LIN {X 0,Y 500.649,Z 462.149,A -85,B 0,C 180,E1 12941.575,E2 12941.575} C_VEL
LIN {X 0,Y 506.783,Z 470.16,A -85,B 0,C 180,E1 12939.56,E2 12939.56} C_VEL
LIN {X 0,Y 513.337,Z 479.72,A -85,B 0,C 180,E1 12937.586,E2 12937.586} C_VEL
LIN {X 0,Y 523.821,Z 496.267,A -85,B 0,C 180,E1 12934.746,E2 12934.746} C_VEL
LIN {X 0,Y 529.057,Z 505.232,A -85,B 0,C 180,E1 12933.44,E2 12933.44} C_VEL
LIN {X 0,Y 516.289,Z 720.849,A -85,B 0,C 180,E1 12930.101,E2 12930.101} C_VEL
LIN {X 0,Y 510.116,Z 825.661,A -85,B 0,C 180,E1 12928.464,E2 12928.464} C_VEL
LIN {X 0,Y 507.28,Z 853.259,A -85,B 0,C 180,E1 12927.934,E2 12927.934} C_VEL
LIN {X 0,Y 503.396,Z 879.439,A -85,B 0,C 180,E1 12927.252,E2 12927.252} C_VEL
LIN {X 0,Y 499.633,Z 900.65,A -85,B 0,C 180,E1 12926.565,E2 12926.565} C_VEL
LIN {X 0,Y 495.492,Z 920.963,A -85,B 0,C 180,E1 12925.777,E2 12925.777} C_VEL
LIN {X 0,Y 490.621,Z 942.152,A -85,B 0,C 180,E1 12924.809,E2 12924.809} C_VEL
LIN {X 0,Y 484.197,Z 967.245,A -85,B 0,C 180,E1 12923.446,E2 12923.446} C_VEL
LIN {X 0,Y 477.712,Z 989.541,A -85,B 0,C 180,E1 12922.003,E2 12922.003} C_VEL
LIN {X 0,Y 471.761,Z 1008.579,A -85,B 0,C 180,E1 12920.583,E2 12920.583} C_VEL
LIN {X 0,Y 465.626,Z 1027.087,A -85,B 0,C 180,E1 12919.009,E2 12919.009} C_VEL
LIN {X 0,Y 458.527,Z 1047.528,A -85,B 0,C 180,E1 12917.018,E2 12917.018} C_VEL
LIN {X 0,Y 450.725,Z 1068.736,A -85,B 0,C 180,E1 12914.593,E2 12914.593} C_VEL
LIN {X 0,Y 444.621,Z 1084.894,A -85,B 0,C 180,E1 12912.47,E2 12912.47} C_VEL
LIN {X 0,Y 438.714,Z 1100.381,A -85,B 0,C 180,E1 12910.165,E2 12910.165} C_VEL
LIN {X 0,Y 432.278,Z 1117.401,A -85,B 0,C 180,E1 12907.279,E2 12907.279} C_VEL
LIN {X 0,Y 426.222,Z 1133.289,A -85,B 0,C 180,E1 12904.103,E2 12904.103} C_VEL
LIN {X 0,Y 422.001,Z 1145.022,A -85,B 0,C 180,E1 12901.417,E2 12901.417} C_VEL
LIN {X 0,Y 418.256,Z 1156.002,A -85,B 0,C 180,E1 12898.563,E2 12898.563} C_VEL
LIN {X 0,Y 414.556,Z 1167.99,A -85,B 0,C 180,E1 12894.967,E2 12894.967} C_VEL
LIN {X 0,Y 411.822,Z 1177.9,A -85,B 0,C 180,E1 12891.358,E2 12891.358} C_VEL
LIN {X 0,Y 410.259,Z 1184.648,A -85,B 0,C 180,E1 12888.472,E2 12888.472} C_VEL
LIN {X 0,Y 409.201,Z 1190.344,A -85,B 0,C 180,E1 12885.592,E2 12885.592} C_VEL
LIN {X 0,Y 408.507,Z 1195.031,A -85,B 0,C 180,E1 12882.726,E2 12882.726} C_VEL
LIN {X 0,Y 408.142,Z 1198.741,A -85,B 0,C 180,E1 12879.875,E2 12879.875} C_VEL
LIN {X 0,Y 407.972,Z 1201.501,A -85,B 0,C 180,E1 12877.039,E2 12877.039} C_VEL
LIN {X 0,Y 407.917,Z 1203.331,A -85,B 0,C 180,E1 12874.218,E2 12874.218} C_VEL
LIN {X 0,Y 407.911,Z 1204.221,A -85,B 0,C 180,E1 12871.546,E2 12871.546} C_VEL
LIN {X 0,Y 407.912,Z 1204.288,A -85,B 0,C 180,E1 12868.877,E2 12868.877} C_VEL
LIN {X 0,Y 407.916,Z 1203.463,A -85,B 0,C 180,E1 12866.065,E2 12866.065} C_VEL
LIN {X 0,Y 407.964,Z 1201.721,A -85,B 0,C 180,E1 12863.244,E2 12863.244} C_VEL
LIN {X 0,Y 408.116,Z 1199.054,A -85,B 0,C 180,E1 12860.41,E2 12860.41} C_VEL
LIN {X 0,Y 408.484,Z 1195.239,A -85,B 0,C 180,E1 12857.418,E2 12857.418} C_VEL
LIN {X 0,Y 409.157,Z 1190.625,A -85,B 0,C 180,E1 12854.552,E2 12854.552} C_VEL
LIN {X 0,Y 410.263,Z 1184.721,A -85,B 0,C 180,E1 12851.529,E2 12851.529} C_VEL
LIN {X 0,Y 412.02,Z 1177.346,A -85,B 0,C 180,E1 12848.355,E2 12848.355} C_VEL
LIN {X 0,Y 415.114,Z 1166.541,A -85,B 0,C 180,E1 12844.46,E2 12844.46} C_VEL
LIN {X 0,Y 418.676,Z 1155.593,A -85,B 0,C 180,E1 12841.158,E2 12841.158} C_VEL
LIN {X 0,Y 422.528,Z 1144.786,A -85,B 0,C 180,E1 12838.309,E2 12838.309} C_VEL
LIN {X 0,Y 427.171,Z 1132.591,A -85,B 0,C 180,E1 12835.481,E2 12835.481} C_VEL
LIN {X 0,Y 433.755,Z 1116.189,A -85,B 0,C 180,E1 12832.182,E2 12832.182} C_VEL
LIN {X 0,Y 440.101,Z 1100.481,A -85,B 0,C 180,E1 12829.477,E2 12829.477} C_VEL
LIN {X 0,Y 446.32,Z 1085.225,A -85,B 0,C 180,E1 12827.163,E2 12827.163} C_VEL
LIN {X 0,Y 452.763,Z 1069.315,A -85,B 0,C 180,E1 12825.035,E2 12825.035} C_VEL
LIN {X 0,Y 460.874,Z 1048.953,A -85,B 0,C 180,E1 12822.654,E2 12822.654} C_VEL
LIN {X 0,Y 468.875,Z 1027.549,A -85,B 0,C 180,E1 12820.538,E2 12820.538} C_VEL
LIN {X 0,Y 475.563,Z 1008.838,A -85,B 0,C 180,E1 12818.93,E2 12818.93} C_VEL
LIN {X 0,Y 482.02,Z 989.698,A -85,B 0,C 180,E1 12817.493,E2 12817.493} C_VEL
LIN {X 0,Y 489.336,Z 966.442,A -85,B 0,C 180,E1 12815.987,E2 12815.987} C_VEL
LIN {X 0,Y 496.05,Z 942.158,A -85,B 0,C 180,E1 12814.676,E2 12814.676} C_VEL
LIN {X 0,Y 501.27,Z 921.153,A -85,B 0,C 180,E1 12813.719,E2 12813.719} C_VEL
LIN {X 0,Y 505.768,Z 900.797,A -85,B 0,C 180,E1 12812.934,E2 12812.934} C_VEL
LIN {X 0,Y 509.793,Z 879.827,A -85,B 0,C 180,E1 12812.258,E2 12812.258} C_VEL
LIN {X 0,Y 513.643,Z 855.953,A -85,B 0,C 180,E1 12811.636,E2 12811.636} C_VEL
LIN {X 0,Y 517.066,Z 826.781,A -85,B 0,C 180,E1 12811.063,E2 12811.063} C_VEL
LIN {X 0,Y 521.805,Z 756.676,A -85,B 0,C 180,E1 12809.953,E2 12809.953} C_VEL
LIN {X 0,Y 536.543,Z 536.341,A -85,B 0,C 180,E1 12806.519,E2 12806.519} C_VEL
LIN {X 0,Y 538.44,Z 508.698,A -85,B 0,C 180,E1 12806.082,E2 12806.082} C_VEL
LIN {X 0,Y 531.522,Z 497.374,A -85,B 0,C 180,E1 12803.91,E2 12803.91} C_VEL
LIN {X 0,Y 523.953,Z 485.597,A -85,B 0,C 180,E1 12801.201,E2 12801.201} C_VEL
LIN {X 0,Y 519.684,Z 479.746,A -85,B 0,C 180,E1 12799.481,E2 12799.481} C_VEL
LIN {X 0,Y 516.251,Z 475.069,A -85,B 0,C 180,E1 12797.936,E2 12797.936} C_VEL
LIN {X 0,Y 512.607,Z 470.139,A -85,B 0,C 180,E1 12796.08,E2 12796.08} C_VEL
LIN {X 0,Y 508.761,Z 464.995,A -85,B 0,C 180,E1 12793.757,E2 12793.757} C_VEL
LIN {X 0,Y 505.748,Z 461.392,A -85,B 0,C 180,E1 12791.518,E2 12791.518} C_VEL
LIN {X 0,Y 504.696,Z 459.401,A -85,B 0,C 180,E1 12790.502,E2 12790.502} C_VEL
LIN {X 0,Y 501.449,Z 455.939,A -85,B 0,C 180,E1 12786.181,E2 12786.181} C_VEL
LIN {X 0,Y 500.926,Z 453.438,A -85,B 0,C 180,E1 12783.319,E2 12783.319} C_VEL
LIN {X 0,Y 500.952,Z 453.714,A -85,B 0,C 180,E1 12781.945,E2 12781.945} C_VEL
LIN {X 0,Y 503.821,Z 458.829,A -85,B 0,C 180,E1 12776.131,E2 12776.131} C_VEL
LIN {X 0,Y 504.993,Z 459.862,A -85,B 0,C 180,E1 12775.002,E2 12775.002} C_VEL
LIN {X 0,Y 507.681,Z 463.98,A -85,B 0,C 180,E1 12772.759,E2 12772.759} C_VEL
LIN {X 0,Y 509.358,Z 465.743,A -85,B 0,C 180,E1 12771.647,E2 12771.647} C_VEL
LIN {X 0,Y 512.705,Z 470.216,A -85,B 0,C 180,E1 12769.664,E2 12769.664} C_VEL
LIN {X 0,Y 517.641,Z 476.786,A -85,B 0,C 180,E1 12767.222,E2 12767.222} C_VEL
LIN {X 0,Y 522.414,Z 483.411,A -85,B 0,C 180,E1 12765.196,E2 12765.196} C_VEL
LIN {X 0,Y 527.766,Z 490.712,A -85,B 0,C 180,E1 12763.206,E2 12763.206} C_VEL
LIN {X 0,Y 535.807,Z 502.584,A -85,B 0,C 180,E1 12760.571,E2 12760.571} C_VEL
LIN {X 0,Y 538.454,Z 506.775,A -85,B 0,C 180,E1 12759.773,E2 12759.773} C_VEL
LIN {X 0,Y 524.368,Z 714.828,A -85,B 0,C 180,E1 12756.529,E2 12756.529} C_VEL
LIN {X 0,Y 517.356,Z 819.989,A -85,B 0,C 180,E1 12754.874,E2 12754.874} C_VEL
LIN {X 0,Y 514.276,Z 847.618,A -85,B 0,C 180,E1 12754.34,E2 12754.34} C_VEL
LIN {X 0,Y 510.217,Z 873.27,A -85,B 0,C 180,E1 12753.669,E2 12753.669} C_VEL
LIN {X 0,Y 506.139,Z 894.675,A -85,B 0,C 180,E1 12752.975,E2 12752.975} C_VEL
LIN {X 0,Y 501.675,Z 915.064,A -85,B 0,C 180,E1 12752.18,E2 12752.18} C_VEL
LIN {X 0,Y 496.561,Z 935.717,A -85,B 0,C 180,E1 12751.232,E2 12751.232} C_VEL
LIN {X 0,Y 489.92,Z 959.881,A -85,B 0,C 180,E1 12749.92,E2 12749.92} C_VEL
LIN {X 0,Y 482.807,Z 982.517,A -85,B 0,C 180,E1 12748.451,E2 12748.451} C_VEL
LIN {X 0,Y 476.282,Z 1001.817,A -85,B 0,C 180,E1 12747,E2 12747} C_VEL
LIN {X 0,Y 469.809,Z 1019.855,A -85,B 0,C 180,E1 12745.449,E2 12745.449} C_VEL
LIN {X 0,Y 462.48,Z 1039.301,A -85,B 0,C 180,E1 12743.538,E2 12743.538} C_VEL
LIN {X 0,Y 453.885,Z 1060.944,A -85,B 0,C 180,E1 12741.043,E2 12741.043} C_VEL
LIN {X 0,Y 447.252,Z 1077.112,A -85,B 0,C 180,E1 12738.884,E2 12738.884} C_VEL
LIN {X 0,Y 441.031,Z 1092.119,A -85,B 0,C 180,E1 12736.61,E2 12736.61} C_VEL
LIN {X 0,Y 434.761,Z 1107.334,A -85,B 0,C 180,E1 12733.99,E2 12733.99} C_VEL
LIN {X 0,Y 427.725,Z 1124.554,A -85,B 0,C 180,E1 12730.531,E2 12730.531} C_VEL
LIN {X 0,Y 423.052,Z 1136.488,A -85,B 0,C 180,E1 12727.744,E2 12727.744} C_VEL
LIN {X 0,Y 419.137,Z 1147.1,A -85,B 0,C 180,E1 12724.926,E2 12724.926} C_VEL
LIN {X 0,Y 415.741,Z 1157.091,A -85,B 0,C 180,E1 12721.897,E2 12721.897} C_VEL
LIN {X 0,Y 412.5,Z 1167.903,A -85,B 0,C 180,E1 12718.05,E2 12718.05} C_VEL
LIN {X 0,Y 410.47,Z 1175.834,A -85,B 0,C 180,E1 12714.616,E2 12714.616} C_VEL
LIN {X 0,Y 409.314,Z 1181.594,A -85,B 0,C 180,E1 12711.645,E2 12711.645} C_VEL
LIN {X 0,Y 408.567,Z 1186.304,A -85,B 0,C 180,E1 12708.698,E2 12708.698} C_VEL
LIN {X 0,Y 408.177,Z 1190.004,A -85,B 0,C 180,E1 12705.777,E2 12705.777} C_VEL
LIN {X 0,Y 407.984,Z 1192.727,A -85,B 0,C 180,E1 12702.886,E2 12702.886} C_VEL
LIN {X 0,Y 407.921,Z 1194.501,A -85,B 0,C 180,E1 12700.022,E2 12700.022} C_VEL
LIN {X 0,Y 407.919,Z 1195.326,A -85,B 0,C 180,E1 12697.322,E2 12697.322} C_VEL
LIN {X 0,Y 407.905,Z 1195.359,A -85,B 0,C 180,E1 12694.803,E2 12694.803} C_VEL
LIN {X 0,Y 406.92,Z 1195.204,A -85,B 0,C 180,E1 12693.721,E2 12693.721} C_VEL
LIN {X 0,Y 401.978,Z 1194.558,A -85,B 0,C 180,E1 12691.527,E2 12691.527} C_VEL
LIN {X 0,Y 400.057,Z 1193.818,A -85,B 0,C 180,E1 12690.199,E2 12690.199} C_VEL
LIN {X 0,Y 399.972,Z 1193.575,A -85,B 0,C 180,E1 12689.88,E2 12689.88} C_VEL
LIN {X 0,Y 400.145,Z 1190.587,A -85,B 0,C 180,E1 12686.418,E2 12686.418} C_VEL
LIN {X 0,Y 400.568,Z 1186.761,A -85,B 0,C 180,E1 12683.262,E2 12683.262} C_VEL
LIN {X 0,Y 401.314,Z 1182.083,A -85,B 0,C 180,E1 12680.245,E2 12680.245} C_VEL
LIN {X 0,Y 402.511,Z 1176.366,A -85,B 0,C 180,E1 12677.227,E2 12677.227} C_VEL
LIN {X 0,Y 404.331,Z 1169.229,A -85,B 0,C 180,E1 12674.068,E2 12674.068} C_VEL
LIN {X 0,Y 407.469,Z 1158.801,A -85,B 0,C 180,E1 12670.206,E2 12670.206} C_VEL
LIN {X 0,Y 411.238,Z 1147.66,A -85,B 0,C 180,E1 12666.792,E2 12666.792} C_VEL
LIN {X 0,Y 415.137,Z 1136.992,A -85,B 0,C 180,E1 12663.949,E2 12663.949} C_VEL
LIN {X 0,Y 419.622,Z 1125.365,A -85,B 0,C 180,E1 12661.227,E2 12661.227} C_VEL
LIN {X 0,Y 425.801,Z 1110.09,A -85,B 0,C 180,E1 12658.105,E2 12658.105} C_VEL
LIN {X 0,Y 432.54,Z 1093.213,A -85,B 0,C 180,E1 12655.181,E2 12655.181} C_VEL
LIN {X 0,Y 438.402,Z 1078.627,A -85,B 0,C 180,E1 12652.965,E2 12652.965} C_VEL
LIN {X 0,Y 444.443,Z 1063.364,A -85,B 0,C 180,E1 12650.911,E2 12650.911} C_VEL
LIN {X 0,Y 450.831,Z 1046.832,A -85,B 0,C 180,E1 12648.946,E2 12648.946} C_VEL
LIN {X 0,Y 458.984,Z 1024.761,A -85,B 0,C 180,E1 12646.668,E2 12646.668} C_VEL
LIN {X 0,Y 465.894,Z 1004.728,A -85,B 0,C 180,E1 12644.909,E2 12644.909} C_VEL
LIN {X 0,Y 471.704,Z 986.875,A -85,B 0,C 180,E1 12643.536,E2 12643.536} C_VEL
LIN {X 0,Y 477.203,Z 968.666,A -85,B 0,C 180,E1 12642.299,E2 12642.299} C_VEL
LIN {X 0,Y 482.904,Z 948.204,A -85,B 0,C 180,E1 12641.089,E2 12641.089} C_VEL
LIN {X 0,Y 489.102,Z 923.711,A -85,B 0,C 180,E1 12639.857,E2 12639.857} C_VEL
LIN {X 0,Y 494.568,Z 898.087,A -85,B 0,C 180,E1 12638.81,E2 12638.81} C_VEL
LIN {X 0,Y 498.547,Z 876.437,A -85,B 0,C 180,E1 12638.082,E2 12638.082} C_VEL
LIN {X 0,Y 501.804,Z 855.388,A -85,B 0,C 180,E1 12637.5,E2 12637.5} C_VEL
LIN {X 0,Y 504.663,Z 832.536,A -85,B 0,C 180,E1 12636.999,E2 12636.999} C_VEL
LIN {X 0,Y 507.414,Z 797.216,A -85,B 0,C 180,E1 12636.402,E2 12636.402} C_VEL
LIN {X 0,Y 520.73,Z 575.134,A -85,B 0,C 180,E1 12632.96,E2 12632.96} C_VEL
LIN {X 0,Y 524.893,Z 506.946,A -85,B 0,C 180,E1 12631.884,E2 12631.884} C_VEL
LIN {X 0,Y 515.61,Z 493.078,A -85,B 0,C 180,E1 12629.475,E2 12629.475} C_VEL
LIN {X 0,Y 507.533,Z 481.415,A -85,B 0,C 180,E1 12627.134,E2 12627.134} C_VEL
LIN {X 0,Y 499.579,Z 470.522,A -85,B 0,C 180,E1 12624.539,E2 12624.539} C_VEL
LIN {X 0,Y 495.044,Z 464.466,A -85,B 0,C 180,E1 12622.881,E2 12622.881} C_VEL
LIN {X 0,Y 492.214,Z 460.736,A -85,B 0,C 180,E1 12621.761,E2 12621.761} C_VEL
LIN {X 0,Y 488.391,Z 455.782,A -85,B 0,C 180,E1 12620.118,E2 12620.118} C_VEL
LIN {X 0,Y 484.466,Z 450.681,A -85,B 0,C 180,E1 12618.221,E2 12618.221} C_VEL
LIN {X 0,Y 481.081,Z 446.451,A -85,B 0,C 180,E1 12616.357,E2 12616.357} C_VEL
LIN {X 0,Y 480.021,Z 445.116,A -85,B 0,C 180,E1 12615.711,E2 12615.711} C_VEL
LIN {X 0,Y 476.73,Z 441.248,A -85,B 0,C 180,E1 12613.463,E2 12613.463} C_VEL
LIN {X 0,Y 475.75,Z 439.436,A -85,B 0,C 180,E1 12612.626,E2 12612.626} C_VEL
LIN {X 0,Y 472.527,Z 436.477,A -85,B 0,C 180,E1 12609.5,E2 12609.5} C_VEL
LIN {X 0,Y 471.237,Z 433.403,A -85,B 0,C 180,E1 12607.314,E2 12607.314} C_VEL
LIN {X 0,Y 470.236,Z 433.066,A -85,B 0,C 180,E1 12601.218,E2 12601.218} C_VEL
LIN {X 0,Y 471.366,Z 433.605,A -85,B 0,C 180,E1 12598.541,E2 12598.541} C_VEL
LIN {X 0,Y 473.121,Z 437.382,A -85,B 0,C 180,E1 12595.879,E2 12595.879} C_VEL
LIN {X 0,Y 476.09,Z 439.999,A -85,B 0,C 180,E1 12593.185,E2 12593.185} C_VEL
LIN {X 0,Y 479.035,Z 444.326,A -85,B 0,C 180,E1 12590.993,E2 12590.993} C_VEL
LIN {X 0,Y 480.77,Z 445.966,A -85,B 0,C 180,E1 12589.939,E2 12589.939} C_VEL
LIN {X 0,Y 484.188,Z 450.411,A -85,B 0,C 180,E1 12588.022,E2 12588.022} C_VEL
LIN {X 0,Y 485.549,Z 452.146,A -85,B 0,C 180,E1 12587.331,E2 12587.331} C_VEL
LIN {X 0,Y 490.234,Z 458.25,A -85,B 0,C 180,E1 12585.169,E2 12585.169} C_VEL
LIN {X 0,Y 494.275,Z 463.516,A -85,B 0,C 180,E1 12583.518,E2 12583.518} C_VEL
LIN {X 0,Y 499.024,Z 469.912,A -85,B 0,C 180,E1 12581.755,E2 12581.755} C_VEL
LIN {X 0,Y 504.843,Z 477.66,A -85,B 0,C 180,E1 12579.811,E2 12579.811} C_VEL
LIN {X 0,Y 511.142,Z 486.977,A -85,B 0,C 180,E1 12577.879,E2 12577.879} C_VEL
LIN {X 0,Y 521.2,Z 503.153,A -85,B 0,C 180,E1 12575.096,E2 12575.096} C_VEL
LIN {X 0,Y 524.916,Z 509.779,A -85,B 0,C 180,E1 12574.136,E2 12574.136} C_VEL
LIN {X 0,Y 511.66,Z 727.256,A -85,B 0,C 180,E1 12570.761,E2 12570.761} C_VEL
LIN {X 0,Y 505.683,Z 825.643,A -85,B 0,C 180,E1 12569.219,E2 12569.219} C_VEL
LIN {X 0,Y 502.773,Z 853.268,A -85,B 0,C 180,E1 12568.688,E2 12568.688} C_VEL
LIN {X 0,Y 498.795,Z 879.444,A -85,B 0,C 180,E1 12568.008,E2 12568.008} C_VEL
LIN {X 0,Y 495.004,Z 900.352,A -85,B 0,C 180,E1 12567.332,E2 12567.332} C_VEL
LIN {X 0,Y 490.612,Z 921.356,A -85,B 0,C 180,E1 12566.519,E2 12566.519} C_VEL
LIN {X 0,Y 485.516,Z 942.93,A -85,B 0,C 180,E1 12565.529,E2 12565.529} C_VEL
LIN {X 0,Y 478.478,Z 969.334,A -85,B 0,C 180,E1 12564.073,E2 12564.073} C_VEL
LIN {X 0,Y 472.363,Z 989.767,A -85,B 0,C 180,E1 12562.741,E2 12562.741} C_VEL
LIN {X 0,Y 466.248,Z 1008.785,A -85,B 0,C 180,E1 12561.316,E2 12561.316} C_VEL
LIN {X 0,Y 459.936,Z 1027.265,A -85,B 0,C 180,E1 12559.735,E2 12559.735} C_VEL
LIN {X 0,Y 452.09,Z 1049.172,A -85,B 0,C 180,E1 12557.579,E2 12557.579} C_VEL
LIN {X 0,Y 444.34,Z 1069.399,A -85,B 0,C 180,E1 12555.224,E2 12555.224} C_VEL
LIN {X 0,Y 438.024,Z 1085.545,A -85,B 0,C 180,E1 12553.074,E2 12553.074} C_VEL
LIN {X 0,Y 431.946,Z 1100.916,A -85,B 0,C 180,E1 12550.752,E2 12550.752} C_VEL
LIN {X 0,Y 425.025,Z 1118.465,A -85,B 0,C 180,E1 12547.71,E2 12547.71} C_VEL
LIN {X 0,Y 419.256,Z 1133.037,A -85,B 0,C 180,E1 12544.75,E2 12544.75} C_VEL
LIN {X 0,Y 414.815,Z 1144.793,A -85,B 0,C 180,E1 12542.026,E2 12542.026} C_VEL
LIN {X 0,Y 411.076,Z 1155.274,A -85,B 0,C 180,E1 12539.269,E2 12539.269} C_VEL
LIN {X 0,Y 407.531,Z 1165.97,A -85,B 0,C 180,E1 12536.052,E2 12536.052} C_VEL
LIN {X 0,Y 404.29,Z 1177.031,A -85,B 0,C 180,E1 12532.082,E2 12532.082} C_VEL
LIN {X 0,Y 402.43,Z 1184.512,A -85,B 0,C 180,E1 12528.845,E2 12528.845} C_VEL
LIN {X 0,Y 401.292,Z 1190.255,A -85,B 0,C 180,E1 12525.889,E2 12525.889} C_VEL
LIN {X 0,Y 400.553,Z 1194.921,A -85,B 0,C 180,E1 12522.983,E2 12522.983} C_VEL
LIN {X 0,Y 400.16,Z 1198.641,A -85,B 0,C 180,E1 12520.074,E2 12520.074} C_VEL
LIN {X 0,Y 399.98,Z 1201.407,A -85,B 0,C 180,E1 12517.181,E2 12517.181} C_VEL
LIN {X 0,Y 399.919,Z 1203.172,A -85,B 0,C 180,E1 12514.446,E2 12514.446} C_VEL
LIN {X 0,Y 399.91,Z 1204.11,A -85,B 0,C 180,E1 12511.72,E2 12511.72} C_VEL
LIN {X 0,Y 399.913,Z 1204.201,A -85,B 0,C 180,E1 12508.854,E2 12508.854} C_VEL
LIN {X 0,Y 399.916,Z 1203.378,A -85,B 0,C 180,E1 12505.986,E2 12505.986} C_VEL
LIN {X 0,Y 399.967,Z 1201.639,A -85,B 0,C 180,E1 12503.109,E2 12503.109} C_VEL
LIN {X 0,Y 400.134,Z 1198.977,A -85,B 0,C 180,E1 12500.217,E2 12500.217} C_VEL
LIN {X 0,Y 400.529,Z 1195.171,A -85,B 0,C 180,E1 12497.164,E2 12497.164} C_VEL
LIN {X 0,Y 401.256,Z 1190.568,A -85,B 0,C 180,E1 12494.24,E2 12494.24} C_VEL
LIN {X 0,Y 402.439,Z 1184.677,A -85,B 0,C 180,E1 12491.157,E2 12491.157} C_VEL
LIN {X 0,Y 404.211,Z 1177.673,A -85,B 0,C 180,E1 12488.068,E2 12488.068} C_VEL
LIN {X 0,Y 407.315,Z 1167.462,A -85,B 0,C 180,E1 12484.247,E2 12484.247} C_VEL
LIN {X 0,Y 411.36,Z 1155.619,A -85,B 0,C 180,E1 12480.595,E2 12480.595} C_VEL
LIN {X 0,Y 415.404,Z 1144.835,A -85,B 0,C 180,E1 12477.701,E2 12477.701} C_VEL
LIN {X 0,Y 420.266,Z 1132.729,A -85,B 0,C 180,E1 12474.848,E2 12474.848} C_VEL
LIN {X 0,Y 426.858,Z 1117.069,A -85,B 0,C 180,E1 12471.631,E2 12471.631} C_VEL
LIN {X 0,Y 434.127,Z 1099.793,A -85,B 0,C 180,E1 12468.624,E2 12468.624} C_VEL
LIN {X 0,Y 440.595,Z 1084.568,A -85,B 0,C 180,E1 12466.306,E2 12466.306} C_VEL
LIN {X 0,Y 447.564,Z 1068.023,A -85,B 0,C 180,E1 12464.091,E2 12464.091} C_VEL
LIN {X 0,Y 456.708,Z 1045.635,A -85,B 0,C 180,E1 12461.519,E2 12461.519} C_VEL
LIN {X 0,Y 463.896,Z 1027.059,A -85,B 0,C 180,E1 12459.694,E2 12459.694} C_VEL
LIN {X 0,Y 470.739,Z 1008.48,A -85,B 0,C 180,E1 12458.098,E2 12458.098} C_VEL
LIN {X 0,Y 477.478,Z 989.056,A -85,B 0,C 180,E1 12456.643,E2 12456.643} C_VEL
LIN {X 0,Y 485.246,Z 964.909,A -85,B 0,C 180,E1 12455.093,E2 12455.093} C_VEL
LIN {X 0,Y 491.829,Z 941.655,A -85,B 0,C 180,E1 12453.852,E2 12453.852} C_VEL
LIN {X 0,Y 497.181,Z 920.632,A -85,B 0,C 180,E1 12452.9,E2 12452.9} C_VEL
LIN {X 0,Y 501.767,Z 900.354,A -85,B 0,C 180,E1 12452.125,E2 12452.125} C_VEL
LIN {X 0,Y 505.982,Z 878.799,A -85,B 0,C 180,E1 12451.436,E2 12451.436} C_VEL
LIN {X 0,Y 510.346,Z 852.054,A -85,B 0,C 180,E1 12450.759,E2 12450.759} C_VEL
LIN {X 0,Y 513.404,Z 824.903,A -85,B 0,C 180,E1 12450.245,E2 12450.245} C_VEL
LIN {X 0,Y 523.571,Z 675.798,A -85,B 0,C 180,E1 12447.904,E2 12447.904} C_VEL
LIN {X 0,Y 534.88,Z 513.617,A -85,B 0,C 180,E1 12445.363,E2 12445.363} C_VEL
LIN {X 0,Y 529.15,Z 504.104,A -85,B 0,C 180,E1 12443.498,E2 12443.498} C_VEL
LIN {X 0,Y 522.018,Z 492.763,A -85,B 0,C 180,E1 12440.871,E2 12440.871} C_VEL
LIN {X 0,Y 518.002,Z 487.199,A -85,B 0,C 180,E1 12439.215,E2 12439.215} C_VEL
LIN {X 0,Y 514.708,Z 482.637,A -85,B 0,C 180,E1 12437.699,E2 12437.699} C_VEL
LIN {X 0,Y 511.234,Z 477.845,A -85,B 0,C 180,E1 12435.892,E2 12435.892} C_VEL
LIN {X 0,Y 507.454,Z 472.745,A -85,B 0,C 180,E1 12433.561,E2 12433.561} C_VEL
LIN {X 0,Y 504.457,Z 468.974,A -85,B 0,C 180,E1 12431.259,E2 12431.259} C_VEL
LIN {X 0,Y 503.607,Z 467.296,A -85,B 0,C 180,E1 12430.409,E2 12430.409} C_VEL
LIN {X 0,Y 500.383,Z 463.724,A -85,B 0,C 180,E1 12425.964,E2 12425.964} C_VEL
LIN {X 0,Y 499.95,Z 461.378,A -85,B 0,C 180,E1 12423.325,E2 12423.325} C_VEL
LIN {X 0,Y 499.967,Z 461.587,A -85,B 0,C 180,E1 12422.063,E2 12422.063} C_VEL
LIN {X 0,Y 502.734,Z 466.712,A -85,B 0,C 180,E1 12416.237,E2 12416.237} C_VEL
LIN {X 0,Y 503.829,Z 467.665,A -85,B 0,C 180,E1 12415.162,E2 12415.162} C_VEL
LIN {X 0,Y 506.541,Z 471.855,A -85,B 0,C 180,E1 12412.856,E2 12412.856} C_VEL
LIN {X 0,Y 508.107,Z 473.573,A -85,B 0,C 180,E1 12411.798,E2 12411.798} C_VEL
LIN {X 0,Y 511.518,Z 478.101,A -85,B 0,C 180,E1 12409.753,E2 12409.753} C_VEL
LIN {X 0,Y 516.396,Z 484.865,A -85,B 0,C 180,E1 12407.304,E2 12407.304} C_VEL
LIN {X 0,Y 520.616,Z 490.752,A -85,B 0,C 180,E1 12405.485,E2 12405.485} C_VEL
LIN {X 0,Y 526.017,Z 498.294,A -85,B 0,C 180,E1 12403.433,E2 12403.433} C_VEL
LIN {X 0,Y 533.794,Z 509.937,A -85,B 0,C 180,E1 12400.836,E2 12400.836} C_VEL
LIN {X 0,Y 534.916,Z 511.854,A -85,B 0,C 180,E1 12400.483,E2 12400.483} C_VEL
LIN {X 0,Y 520.435,Z 719.909,A -85,B 0,C 180,E1 12397.238,E2 12397.238} C_VEL
LIN {X 0,Y 513.544,Z 820.121,A -85,B 0,C 180,E1 12395.659,E2 12395.659} C_VEL
LIN {X 0,Y 510.382,Z 847.808,A -85,B 0,C 180,E1 12395.125,E2 12395.125} C_VEL
LIN {X 0,Y 506.227,Z 873.449,A -85,B 0,C 180,E1 12394.457,E2 12394.457} C_VEL
LIN {X 0,Y 502.215,Z 894.076,A -85,B 0,C 180,E1 12393.794,E2 12393.794} C_VEL
LIN {X 0,Y 497.546,Z 914.911,A -85,B 0,C 180,E1 12392.988,E2 12392.988} C_VEL
LIN {X 0,Y 492.358,Z 935.372,A -85,B 0,C 180,E1 12392.053,E2 12392.053} C_VEL
LIN {X 0,Y 485.431,Z 959.924,A -85,B 0,C 180,E1 12390.727,E2 12390.727} C_VEL
LIN {X 0,Y 478.115,Z 982.557,A -85,B 0,C 180,E1 12389.261,E2 12389.261} C_VEL
LIN {X 0,Y 471.402,Z 1001.847,A -85,B 0,C 180,E1 12387.811,E2 12387.811} C_VEL
LIN {X 0,Y 464.734,Z 1019.886,A -85,B 0,C 180,E1 12386.258,E2 12386.258} C_VEL
LIN {X 0,Y 457.407,Z 1038.698,A -85,B 0,C 180,E1 12384.407,E2 12384.407} C_VEL
LIN {X 0,Y 448.242,Z 1060.991,A -85,B 0,C 180,E1 12381.837,E2 12381.837} C_VEL
LIN {X 0,Y 441.158,Z 1077.609,A -85,B 0,C 180,E1 12379.599,E2 12379.599} C_VEL
LIN {X 0,Y 434.872,Z 1092.177,A -85,B 0,C 180,E1 12377.37,E2 12377.37} C_VEL
LIN {X 0,Y 428.503,Z 1106.952,A -85,B 0,C 180,E1 12374.804,E2 12374.804} C_VEL
LIN {X 0,Y 421.127,Z 1124.251,A -85,B 0,C 180,E1 12371.303,E2 12371.303} C_VEL
LIN {X 0,Y 415.936,Z 1136.803,A -85,B 0,C 180,E1 12368.331,E2 12368.331} C_VEL
LIN {X 0,Y 411.829,Z 1147.385,A -85,B 0,C 180,E1 12365.468,E2 12365.468} C_VEL
LIN {X 0,Y 408.139,Z 1157.678,A -85,B 0,C 180,E1 12362.28,E2 12362.28} C_VEL
LIN {X 0,Y 404.592,Z 1168.833,A -85,B 0,C 180,E1 12358.165,E2 12358.165} C_VEL
LIN {X 0,Y 402.58,Z 1176.329,A -85,B 0,C 180,E1 12354.817,E2 12354.817} C_VEL
LIN {X 0,Y 401.372,Z 1182.017,A -85,B 0,C 180,E1 12351.788,E2 12351.788} C_VEL
LIN {X 0,Y 400.591,Z 1186.659,A -85,B 0,C 180,E1 12348.782,E2 12348.782} C_VEL
LIN {X 0,Y 400.184,Z 1190.294,A -85,B 0,C 180,E1 12345.803,E2 12345.803} C_VEL
LIN {X 0,Y 399.985,Z 1192.956,A -85,B 0,C 180,E1 12342.854,E2 12342.854} C_VEL
LIN {X 0,Y 399.921,Z 1194.685,A -85,B 0,C 180,E1 12339.906,E2 12339.906} C_VEL
LIN {X 0,Y 399.901,Z 1195.486,A -85,B 0,C 180,E1 12336.892,E2 12336.892} C_VEL
LIN {X 0,Y 399.913,Z 1195.258,A -85,B 0,C 180,E1 12333.583,E2 12333.583} C_VEL
LIN {X 0,Y 399.972,Z 1193.575,A -85,B 0,C 180,E1 12329.88,E2 12329.88} C_VEL
LIN {X 0,Y 399.009,Z 1192.776,A -85,B 0,C 180,E1 12328.783,E2 12328.783} C_VEL
LIN {X 0,Y 392.748,Z 1190.081,A -85,B 0,C 180,E1 12325.69,E2 12325.69} C_VEL
LIN {X 0,Y 392.306,Z 1189.224,A -85,B 0,C 180,E1 12324.886,E2 12324.886} C_VEL
LIN {X 0,Y 393.111,Z 1183.833,A -85,B 0,C 180,E1 12320.926,E2 12320.926} C_VEL
LIN {X 0,Y 394.43,Z 1177.539,A -85,B 0,C 180,E1 12317.407,E2 12317.407} C_VEL
LIN {X 0,Y 396.136,Z 1170.921,A -85,B 0,C 180,E1 12314.331,E2 12314.331} C_VEL
LIN {X 0,Y 398.481,Z 1163.181,A -85,B 0,C 180,E1 12311.265,E2 12311.265} C_VEL
LIN {X 0,Y 401.512,Z 1154.26,A -85,B 0,C 180,E1 12308.219,E2 12308.219} C_VEL
LIN {X 0,Y 406.101,Z 1142.068,A -85,B 0,C 180,E1 12304.633,E2 12304.633} C_VEL
LIN {X 0,Y 411.499,Z 1128.295,A -85,B 0,C 180,E1 12301.242,E2 12301.242} C_VEL
LIN {X 0,Y 416.546,Z 1116.038,A -85,B 0,C 180,E1 12298.608,E2 12298.608} C_VEL
LIN {X 0,Y 421.961,Z 1103.139,A -85,B 0,C 180,E1 12296.161,E2 12296.161} C_VEL
LIN {X 0,Y 428.33,Z 1088.018,A -85,B 0,C 180,E1 12293.634,E2 12293.634} C_VEL
LIN {X 0,Y 436.529,Z 1068.21,A -85,B 0,C 180,E1 12290.788,E2 12290.788} C_VEL
LIN {X 0,Y 443.37,Z 1051.113,A -85,B 0,C 180,E1 12288.676,E2 12288.676} C_VEL
LIN {X 0,Y 449.759,Z 1034.555,A -85,B 0,C 180,E1 12286.873,E2 12286.873} C_VEL
LIN {X 0,Y 456.197,Z 1017.112,A -85,B 0,C 180,E1 12285.198,E2 12285.198} C_VEL
LIN {X 0,Y 463.988,Z 994.851,A -85,B 0,C 180,E1 12283.339,E2 12283.339} C_VEL
LIN {X 0,Y 471.365,Z 971.438,A -85,B 0,C 180,E1 12281.696,E2 12281.696} C_VEL
LIN {X 0,Y 477.194,Z 951.273,A -85,B 0,C 180,E1 12280.482,E2 12280.482} C_VEL
LIN {X 0,Y 482.389,Z 931.546,A -85,B 0,C 180,E1 12279.456,E2 12279.456} C_VEL
LIN {X 0,Y 487.438,Z 910.138,A -85,B 0,C 180,E1 12278.503,E2 12278.503} C_VEL
LIN {X 0,Y 493.064,Z 882.255,A -85,B 0,C 180,E1 12277.488,E2 12277.488} C_VEL
LIN {X 0,Y 496.921,Z 858.641,A -85,B 0,C 180,E1 12276.811,E2 12276.811} C_VEL
LIN {X 0,Y 499.788,Z 836.934,A -85,B 0,C 180,E1 12276.318,E2 12276.318} C_VEL
LIN {X 0,Y 501.967,Z 814.298,A -85,B 0,C 180,E1 12275.907,E2 12275.907} C_VEL
LIN {X 0,Y 515.635,Z 594.128,A -85,B 0,C 180,E1 12272.48,E2 12272.48} C_VEL
LIN {X 0,Y 520.868,Z 511.645,A -85,B 0,C 180,E1 12271.187,E2 12271.187} C_VEL
LIN {X 0,Y 511.122,Z 496.952,A -85,B 0,C 180,E1 12268.547,E2 12268.547} C_VEL
LIN {X 0,Y 502.073,Z 483.904,A -85,B 0,C 180,E1 12265.763,E2 12265.763} C_VEL
LIN {X 0,Y 494.357,Z 473.321,A -85,B 0,C 180,E1 12263.033,E2 12263.033} C_VEL
LIN {X 0,Y 490.425,Z 468.133,A -85,B 0,C 180,E1 12261.467,E2 12261.467} C_VEL
LIN {X 0,Y 486.797,Z 463.349,A -85,B 0,C 180,E1 12259.873,E2 12259.873} C_VEL
LIN {X 0,Y 482.821,Z 458.177,A -85,B 0,C 180,E1 12257.911,E2 12257.911} C_VEL
LIN {X 0,Y 479.396,Z 453.585,A -85,B 0,C 180,E1 12255.948,E2 12255.948} C_VEL
LIN {X 0,Y 475.527,Z 449.081,A -85,B 0,C 180,E1 12253.312,E2 12253.312} C_VEL
LIN {X 0,Y 474.487,Z 447.24,A -85,B 0,C 180,E1 12252.412,E2 12252.412} C_VEL
LIN {X 0,Y 471.458,Z 444.366,A -85,B 0,C 180,E1 12249.399,E2 12249.399} C_VEL
LIN {X 0,Y 470.197,Z 441.329,A -85,B 0,C 180,E1 12247.208,E2 12247.208} C_VEL
LIN {X 0,Y 469.29,Z 441.017,A -85,B 0,C 180,E1 12241.099,E2 12241.099} C_VEL
LIN {X 0,Y 470.344,Z 441.601,A -85,B 0,C 180,E1 12238.599,E2 12238.599} C_VEL
LIN {X 0,Y 472.032,Z 445.253,A -85,B 0,C 180,E1 12235.992,E2 12235.992} C_VEL
LIN {X 0,Y 474.883,Z 447.82,A -85,B 0,C 180,E1 12233.35,E2 12233.35} C_VEL
LIN {X 0,Y 477.872,Z 452.205,A -85,B 0,C 180,E1 12231.093,E2 12231.093} C_VEL
LIN {X 0,Y 479.485,Z 453.821,A -85,B 0,C 180,E1 12230.093,E2 12230.093} C_VEL
LIN {X 0,Y 482.982,Z 458.308,A -85,B 0,C 180,E1 12228.113,E2 12228.113} C_VEL
LIN {X 0,Y 488.586,Z 465.784,A -85,B 0,C 180,E1 12225.421,E2 12225.421} C_VEL
LIN {X 0,Y 492.774,Z 471.362,A -85,B 0,C 180,E1 12223.678,E2 12223.678} C_VEL
LIN {X 0,Y 499.365,Z 480.163,A -85,B 0,C 180,E1 12221.254,E2 12221.254} C_VEL
LIN {X 0,Y 506.709,Z 490.681,A -85,B 0,C 180,E1 12218.862,E2 12218.862} C_VEL
LIN {X 0,Y 516.982,Z 507.288,A -85,B 0,C 180,E1 12215.884,E2 12215.884} C_VEL
LIN {X 0,Y 520.862,Z 514.196,A -85,B 0,C 180,E1 12214.844,E2 12214.844} C_VEL
LIN {X 0,Y 507.158,Z 732.706,A -85,B 0,C 180,E1 12211.448,E2 12211.448} C_VEL
LIN {X 0,Y 501.321,Z 825.786,A -85,B 0,C 180,E1 12209.984,E2 12209.984} C_VEL
LIN {X 0,Y 498.305,Z 853.599,A -85,B 0,C 180,E1 12209.447,E2 12209.447} C_VEL
LIN {X 0,Y 494.287,Z 879.416,A -85,B 0,C 180,E1 12208.779,E2 12208.779} C_VEL
LIN {X 0,Y 490.313,Z 900.799,A -85,B 0,C 180,E1 12208.087,E2 12208.087} C_VEL
LIN {X 0,Y 485.815,Z 921.731,A -85,B 0,C 180,E1 12207.274,E2 12207.274} C_VEL
LIN {X 0,Y 480.133,Z 945.122,A -85,B 0,C 180,E1 12206.194,E2 12206.194} C_VEL
LIN {X 0,Y 473.003,Z 970.808,A -85,B 0,C 180,E1 12204.753,E2 12204.753} C_VEL
LIN {X 0,Y 466.976,Z 990.355,A -85,B 0,C 180,E1 12203.469,E2 12203.469} C_VEL
LIN {X 0,Y 460.814,Z 1008.972,A -85,B 0,C 180,E1 12202.067,E2 12202.067} C_VEL
LIN {X 0,Y 454.349,Z 1027.37,A -85,B 0,C 180,E1 12200.485,E2 12200.485} C_VEL
LIN {X 0,Y 446.418,Z 1048.829,A -85,B 0,C 180,E1 12198.364,E2 12198.364} C_VEL
LIN {X 0,Y 438.447,Z 1068.977,A -85,B 0,C 180,E1 12196.01,E2 12196.01} C_VEL
LIN {X 0,Y 432.008,Z 1084.874,A -85,B 0,C 180,E1 12193.884,E2 12193.884} C_VEL
LIN {X 0,Y 425.914,Z 1099.717,A -85,B 0,C 180,E1 12191.635,E2 12191.635} C_VEL
LIN {X 0,Y 419.273,Z 1115.9,A -85,B 0,C 180,E1 12188.844,E2 12188.844} C_VEL
LIN {X 0,Y 412.624,Z 1132.129,A -85,B 0,C 180,E1 12185.562,E2 12185.562} C_VEL
LIN {X 0,Y 407.856,Z 1144.115,A -85,B 0,C 180,E1 12182.765,E2 12182.765} C_VEL
LIN {X 0,Y 403.853,Z 1154.758,A -85,B 0,C 180,E1 12179.939,E2 12179.939} C_VEL
LIN {X 0,Y 400.319,Z 1164.842,A -85,B 0,C 180,E1 12176.878,E2 12176.878} C_VEL
LIN {X 0,Y 396.908,Z 1175.793,A -85,B 0,C 180,E1 12172.984,E2 12172.984} C_VEL
LIN {X 0,Y 394.694,Z 1184.06,A -85,B 0,C 180,E1 12169.382,E2 12169.382} C_VEL
LIN {X 0,Y 393.4,Z 1190.092,A -85,B 0,C 180,E1 12166.236,E2 12166.236} C_VEL
LIN {X 0,Y 392.607,Z 1194.802,A -85,B 0,C 180,E1 12163.251,E2 12163.251} C_VEL
LIN {X 0,Y 392.173,Z 1198.607,A -85,B 0,C 180,E1 12160.213,E2 12160.213} C_VEL
LIN {X 0,Y 391.989,Z 1201.307,A -85,B 0,C 180,E1 12157.328,E2 12157.328} C_VEL
LIN {X 0,Y 391.92,Z 1203.078,A -85,B 0,C 180,E1 12154.537,E2 12154.537} C_VEL
LIN {X 0,Y 391.91,Z 1204.02,A -85,B 0,C 180,E1 12151.755,E2 12151.755} C_VEL
LIN {X 0,Y 391.914,Z 1204.115,A -85,B 0,C 180,E1 12148.831,E2 12148.831} C_VEL
LIN {X 0,Y 391.916,Z 1203.297,A -85,B 0,C 180,E1 12145.904,E2 12145.904} C_VEL
LIN {X 0,Y 391.976,Z 1201.501,A -85,B 0,C 180,E1 12142.888,E2 12142.888} C_VEL
LIN {X 0,Y 392.167,Z 1198.747,A -85,B 0,C 180,E1 12139.868,E2 12139.868} C_VEL
LIN {X 0,Y 392.58,Z 1195.112,A -85,B 0,C 180,E1 12136.899,E2 12136.899} C_VEL
LIN {X 0,Y 393.361,Z 1190.518,A -85,B 0,C 180,E1 12133.914,E2 12133.914} C_VEL
LIN {X 0,Y 394.632,Z 1184.643,A -85,B 0,C 180,E1 12130.77,E2 12130.77} C_VEL
LIN {X 0,Y 396.52,Z 1177.654,A -85,B 0,C 180,E1 12127.62,E2 12127.62} C_VEL
LIN {X 0,Y 399.806,Z 1167.471,A -85,B 0,C 180,E1 12123.727,E2 12123.727} C_VEL
LIN {X 0,Y 404.072,Z 1155.644,A -85,B 0,C 180,E1 12120.008,E2 12120.008} C_VEL
LIN {X 0,Y 408.338,Z 1144.893,A -85,B 0,C 180,E1 12117.072,E2 12117.072} C_VEL
LIN {X 0,Y 413.166,Z 1133.439,A -85,B 0,C 180,E1 12114.323,E2 12114.323} C_VEL
LIN {X 0,Y 419.675,Z 1118.598,A -85,B 0,C 180,E1 12111.201,E2 12111.201} C_VEL
LIN {X 0,Y 427.529,Z 1100.786,A -85,B 0,C 180,E1 12108.02,E2 12108.02} C_VEL
LIN {X 0,Y 434.451,Z 1085.13,A -85,B 0,C 180,E1 12105.602,E2 12105.602} C_VEL
LIN {X 0,Y 441.328,Z 1069.395,A -85,B 0,C 180,E1 12103.467,E2 12103.467} C_VEL
LIN {X 0,Y 449.859,Z 1049.465,A -85,B 0,C 180,E1 12101.109,E2 12101.109} C_VEL
LIN {X 0,Y 458.454,Z 1028.049,A -85,B 0,C 180,E1 12098.967,E2 12098.967} C_VEL
LIN {X 0,Y 465.484,Z 1009.587,A -85,B 0,C 180,E1 12097.367,E2 12097.367} C_VEL
LIN {X 0,Y 472.305,Z 990.553,A -85,B 0,C 180,E1 12095.929,E2 12095.929} C_VEL
LIN {X 0,Y 479.203,Z 969.903,A -85,B 0,C 180,E1 12094.58,E2 12094.58} C_VEL
LIN {X 0,Y 487.103,Z 943.442,A -85,B 0,C 180,E1 12093.124,E2 12093.124} C_VEL
LIN {X 0,Y 492.889,Z 921.381,A -85,B 0,C 180,E1 12092.121,E2 12092.121} C_VEL
LIN {X 0,Y 497.582,Z 901.229,A -85,B 0,C 180,E1 12091.349,E2 12091.349} C_VEL
LIN {X 0,Y 501.826,Z 880.195,A -85,B 0,C 180,E1 12090.674,E2 12090.674} C_VEL
LIN {X 0,Y 505.731,Z 857.225,A -85,B 0,C 180,E1 12090.079,E2 12090.079} C_VEL
LIN {X 0,Y 509.501,Z 827.079,A -85,B 0,C 180,E1 12089.484,E2 12089.484} C_VEL
LIN {X 0,Y 514.098,Z 763.321,A -85,B 0,C 180,E1 12088.471,E2 12088.471} C_VEL
LIN {X 0,Y 529.758,Z 542.04,A -85,B 0,C 180,E1 12085.021,E2 12085.021} C_VEL
LIN {X 0,Y 531.425,Z 518.456,A -85,B 0,C 180,E1 12084.636,E2 12084.636} C_VEL
LIN {X 0,Y 524.047,Z 506.264,A -85,B 0,C 180,E1 12082.079,E2 12082.079} C_VEL
LIN {X 0,Y 519.308,Z 498.849,A -85,B 0,C 180,E1 12080.219,E2 12080.219} C_VEL
LIN {X 0,Y 515.688,Z 493.779,A -85,B 0,C 180,E1 12078.659,E2 12078.659} C_VEL
LIN {X 0,Y 513.174,Z 490.203,A -85,B 0,C 180,E1 12077.461,E2 12077.461} C_VEL
LIN {X 0,Y 509.766,Z 485.444,A -85,B 0,C 180,E1 12075.647,E2 12075.647} C_VEL
LIN {X 0,Y 506.153,Z 480.49,A -85,B 0,C 180,E1 12073.364,E2 12073.364} C_VEL
LIN {X 0,Y 503.23,Z 476.662,A -85,B 0,C 180,E1 12071.049,E2 12071.049} C_VEL
LIN {X 0,Y 502.397,Z 475.124,A -85,B 0,C 180,E1 12070.203,E2 12070.203} C_VEL
LIN {X 0,Y 499.287,Z 471.402,A -85,B 0,C 180,E1 12065.631,E2 12065.631} C_VEL
LIN {X 0,Y 498.974,Z 469.318,A -85,B 0,C 180,E1 12063.332,E2 12063.332} C_VEL
LIN {X 0,Y 498.985,Z 469.569,A -85,B 0,C 180,E1 12062.067,E2 12062.067} C_VEL
LIN {X 0,Y 501.648,Z 474.595,A -85,B 0,C 180,E1 12056.343,E2 12056.343} C_VEL
LIN {X 0,Y 502.721,Z 475.592,A -85,B 0,C 180,E1 12055.265,E2 12055.265} C_VEL
LIN {X 0,Y 505.559,Z 479.893,A -85,B 0,C 180,E1 12052.842,E2 12052.842} C_VEL
LIN {X 0,Y 506.861,Z 481.4,A -85,B 0,C 180,E1 12051.948,E2 12051.948} C_VEL
LIN {X 0,Y 510.331,Z 485.986,A -85,B 0,C 180,E1 12049.843,E2 12049.843} C_VEL
LIN {X 0,Y 514.925,Z 492.571,A -85,B 0,C 180,E1 12047.496,E2 12047.496} C_VEL
LIN {X 0,Y 519.218,Z 498.652,A -85,B 0,C 180,E1 12045.616,E2 12045.616} C_VEL
LIN {X 0,Y 524.277,Z 505.872,A -85,B 0,C 180,E1 12043.662,E2 12043.662} C_VEL
LIN {X 0,Y 531.464,Z 516.796,A -85,B 0,C 180,E1 12041.207,E2 12041.207} C_VEL
LIN {X 0,Y 517.107,Z 717.427,A -85,B 0,C 180,E1 12038.076,E2 12038.076} C_VEL
LIN {X 0,Y 509.843,Z 820.181,A -85,B 0,C 180,E1 12036.457,E2 12036.457} C_VEL
LIN {X 0,Y 506.625,Z 847.789,A -85,B 0,C 180,E1 12035.926,E2 12035.926} C_VEL
LIN {X 0,Y 502.352,Z 873.541,A -85,B 0,C 180,E1 12035.261,E2 12035.261} C_VEL
LIN {X 0,Y 498.152,Z 894.612,A -85,B 0,C 180,E1 12034.584,E2 12034.584} C_VEL
LIN {X 0,Y 493.353,Z 915.459,A -85,B 0,C 180,E1 12033.779,E2 12033.779} C_VEL
LIN {X 0,Y 487.757,Z 936.918,A -85,B 0,C 180,E1 12032.797,E2 12032.797} C_VEL
LIN {X 0,Y 480.157,Z 962.663,A -85,B 0,C 180,E1 12031.382,E2 12031.382} C_VEL
LIN {X 0,Y 473.233,Z 983.438,A -85,B 0,C 180,E1 12030.027,E2 12030.027} C_VEL
LIN {X 0,Y 466.344,Z 1002.651,A -85,B 0,C 180,E1 12028.576,E2 12028.576} C_VEL
LIN {X 0,Y 459.627,Z 1020.256,A -85,B 0,C 180,E1 12027.053,E2 12027.053} C_VEL
LIN {X 0,Y 451.691,Z 1039.987,A -85,B 0,C 180,E1 12025.099,E2 12025.099} C_VEL
LIN {X 0,Y 442.715,Z 1061.003,A -85,B 0,C 180,E1 12022.654,E2 12022.654} C_VEL
LIN {X 0,Y 435.354,Z 1077.64,A -85,B 0,C 180,E1 12020.401,E2 12020.401} C_VEL
LIN {X 0,Y 428.621,Z 1092.64,A -85,B 0,C 180,E1 12018.086,E2 12018.086} C_VEL
LIN {X 0,Y 421.257,Z 1109.105,A -85,B 0,C 180,E1 12015.174,E2 12015.174} C_VEL
LIN {X 0,Y 414.012,Z 1125.256,A -85,B 0,C 180,E1 12011.802,E2 12011.802} C_VEL
LIN {X 0,Y 408.871,Z 1137.127,A -85,B 0,C 180,E1 12008.937,E2 12008.937} C_VEL
LIN {X 0,Y 404.558,Z 1147.678,A -85,B 0,C 180,E1 12006.03,E2 12006.03} C_VEL
LIN {X 0,Y 400.349,Z 1158.881,A -85,B 0,C 180,E1 12002.476,E2 12002.476} C_VEL
LIN {X 0,Y 396.8,Z 1169.411,A -85,B 0,C 180,E1 11998.44,E2 11998.44} C_VEL
LIN {X 0,Y 394.777,Z 1176.523,A -85,B 0,C 180,E1 11995.182,E2 11995.182} C_VEL
LIN {X 0,Y 393.487,Z 1182.191,A -85,B 0,C 180,E1 11992.09,E2 11992.09} C_VEL
LIN {X 0,Y 392.642,Z 1186.813,A -85,B 0,C 180,E1 11989.023,E2 11989.023} C_VEL
LIN {X 0,Y 392.192,Z 1190.592,A -85,B 0,C 180,E1 11985.83,E2 11985.83} C_VEL
LIN {X 0,Y 391.976,Z 1193.419,A -85,B 0,C 180,E1 11982.522,E2 11982.522} C_VEL
LIN {X 0,Y 391.92,Z 1195.311,A -85,B 0,C 180,E1 11978.657,E2 11978.657} C_VEL
LIN {X 0,Y 391.905,Z 1195.588,A -85,B 0,C 180,E1 11975.123,E2 11975.123} C_VEL
LIN {X 0,Y 391.925,Z 1194.809,A -85,B 0,C 180,E1 11972.046,E2 11972.046} C_VEL
LIN {X 0,Y 391.987,Z 1193.164,A -85,B 0,C 180,E1 11969.123,E2 11969.123} C_VEL
LIN {X 0,Y 392.18,Z 1190.472,A -85,B 0,C 180,E1 11966.052,E2 11966.052} C_VEL
LIN {X 0,Y 392.306,Z 1189.224,A -85,B 0,C 180,E1 11964.886,E2 11964.886} C_VEL
LIN {X 0,Y 391.48,Z 1187.991,A -85,B 0,C 180,E1 11963.773,E2 11963.773} C_VEL
LIN {X 0,Y 385.834,Z 1184.013,A -85,B 0,C 180,E1 11960.717,E2 11960.717} C_VEL
LIN {X 0,Y 385.467,Z 1182.576,A -85,B 0,C 180,E1 11959.831,E2 11959.831} C_VEL
LIN {X 0,Y 386.78,Z 1176.931,A -85,B 0,C 180,E1 11956.698,E2 11956.698} C_VEL
LIN {X 0,Y 388.678,Z 1170.194,A -85,B 0,C 180,E1 11953.562,E2 11953.562} C_VEL
LIN {X 0,Y 391.354,Z 1161.937,A -85,B 0,C 180,E1 11950.29,E2 11950.29} C_VEL
LIN {X 0,Y 395.762,Z 1149.995,A -85,B 0,C 180,E1 11946.315,E2 11946.315} C_VEL
LIN {X 0,Y 400.316,Z 1138.47,A -85,B 0,C 180,E1 11943.088,E2 11943.088} C_VEL
LIN {X 0,Y 405.169,Z 1126.894,A -85,B 0,C 180,E1 11940.262,E2 11940.262} C_VEL
LIN {X 0,Y 410.845,Z 1113.796,A -85,B 0,C 180,E1 11937.462,E2 11937.462} C_VEL
LIN {X 0,Y 418.286,Z 1096.799,A -85,B 0,C 180,E1 11934.319,E2 11934.319} C_VEL
LIN {X 0,Y 425.54,Z 1079.893,A -85,B 0,C 180,E1 11931.661,E2 11931.661} C_VEL
LIN {X 0,Y 432.105,Z 1064.407,A -85,B 0,C 180,E1 11929.528,E2 11929.528} C_VEL
LIN {X 0,Y 438.956,Z 1047.797,A -85,B 0,C 180,E1 11927.516,E2 11927.516} C_VEL
LIN {X 0,Y 447.226,Z 1026.941,A -85,B 0,C 180,E1 11925.314,E2 11925.314} C_VEL
LIN {X 0,Y 455.229,Z 1005.005,A -85,B 0,C 180,E1 11923.363,E2 11923.363} C_VEL
LIN {X 0,Y 461.639,Z 986.355,A -85,B 0,C 180,E1 11921.927,E2 11921.927} C_VEL
LIN {X 0,Y 467.591,Z 967.658,A -85,B 0,C 180,E1 11920.665,E2 11920.665} C_VEL
LIN {X 0,Y 473.755,Z 946.498,A -85,B 0,C 180,E1 11919.425,E2 11919.425} C_VEL
LIN {X 0,Y 480.845,Z 919.02,A -85,B 0,C 180,E1 11918.088,E2 11918.088} C_VEL
LIN {X 0,Y 485.776,Z 896.67,A -85,B 0,C 180,E1 11917.196,E2 11917.196} C_VEL
LIN {X 0,Y 489.82,Z 875.507,A -85,B 0,C 180,E1 11916.496,E2 11916.496} C_VEL
LIN {X 0,Y 493.266,Z 853.964,A -85,B 0,C 180,E1 11915.91,E2 11915.91} C_VEL
LIN {X 0,Y 496.731,Z 826.599,A -85,B 0,C 180,E1 11915.333,E2 11915.333} C_VEL
LIN {X 0,Y 499.863,Z 781.853,A -85,B 0,C 180,E1 11914.611,E2 11914.611} C_VEL
LIN {X 0,Y 513.817,Z 563.217,A -85,B 0,C 180,E1 11911.209,E2 11911.209} C_VEL
LIN {X 0,Y 516.821,Z 516.307,A -85,B 0,C 180,E1 11910.457,E2 11910.457} C_VEL
LIN {X 0,Y 508.135,Z 503.063,A -85,B 0,C 180,E1 11908.022,E2 11908.022} C_VEL
LIN {X 0,Y 499.871,Z 490.974,A -85,B 0,C 180,E1 11905.408,E2 11905.408} C_VEL
LIN {X 0,Y 492.531,Z 480.725,A -85,B 0,C 180,E1 11902.752,E2 11902.752} C_VEL
LIN {X 0,Y 488.382,Z 475.194,A -85,B 0,C 180,E1 11901.058,E2 11901.058} C_VEL
LIN {X 0,Y 485.088,Z 470.778,A -85,B 0,C 180,E1 11899.57,E2 11899.57} C_VEL
LIN {X 0,Y 481.415,Z 465.882,A -85,B 0,C 180,E1 11897.715,E2 11897.715} C_VEL
LIN {X 0,Y 478.002,Z 461.235,A -85,B 0,C 180,E1 11895.717,E2 11895.717} C_VEL
LIN {X 0,Y 474.256,Z 456.782,A -85,B 0,C 180,E1 11893.1,E2 11893.1} C_VEL
LIN {X 0,Y 473.23,Z 455.039,A -85,B 0,C 180,E1 11892.198,E2 11892.198} C_VEL
LIN {X 0,Y 470.304,Z 452.1,A -85,B 0,C 180,E1 11889.175,E2 11889.175} C_VEL
LIN {X 0,Y 469.159,Z 449.254,A -85,B 0,C 180,E1 11887.101,E2 11887.101} C_VEL
LIN {X 0,Y 468.345,Z 448.968,A -85,B 0,C 180,E1 11880.979,E2 11880.979} C_VEL
LIN {X 0,Y 469.273,Z 449.39,A -85,B 0,C 180,E1 11878.779,E2 11878.779} C_VEL
LIN {X 0,Y 470.945,Z 453.125,A -85,B 0,C 180,E1 11876.104,E2 11876.104} C_VEL
LIN {X 0,Y 473.744,Z 455.778,A -85,B 0,C 180,E1 11873.456,E2 11873.456} C_VEL
LIN {X 0,Y 476.71,Z 460.084,A -85,B 0,C 180,E1 11871.192,E2 11871.192} C_VEL
LIN {X 0,Y 478.203,Z 461.668,A -85,B 0,C 180,E1 11870.249,E2 11870.249} C_VEL
LIN {X 0,Y 481.778,Z 466.203,A -85,B 0,C 180,E1 11868.204,E2 11868.204} C_VEL
LIN {X 0,Y 487.198,Z 473.687,A -85,B 0,C 180,E1 11865.56,E2 11865.56} C_VEL
LIN {X 0,Y 490.932,Z 478.704,A -85,B 0,C 180,E1 11863.98,E2 11863.98} C_VEL
LIN {X 0,Y 497.493,Z 487.638,A -85,B 0,C 180,E1 11861.515,E2 11861.515} C_VEL
LIN {X 0,Y 504.573,Z 497.929,A -85,B 0,C 180,E1 11859.163,E2 11859.163} C_VEL
LIN {X 0,Y 514.703,Z 514.627,A -85,B 0,C 180,E1 11856.167,E2 11856.167} C_VEL
LIN {X 0,Y 516.877,Z 518.737,A -85,B 0,C 180,E1 11855.562,E2 11855.562} C_VEL
LIN {X 0,Y 502.843,Z 736.292,A -85,B 0,C 180,E1 11852.176,E2 11852.176} C_VEL
LIN {X 0,Y 497.057,Z 825.806,A -85,B 0,C 180,E1 11850.765,E2 11850.765} C_VEL
LIN {X 0,Y 493.944,Z 853.762,A -85,B 0,C 180,E1 11850.224,E2 11850.224} C_VEL
LIN {X 0,Y 489.848,Z 879.483,A -85,B 0,C 180,E1 11849.56,E2 11849.56} C_VEL
LIN {X 0,Y 485.864,Z 900.477,A -85,B 0,C 180,E1 11848.882,E2 11848.882} C_VEL
LIN {X 0,Y 481.407,Z 920.792,A -85,B 0,C 180,E1 11848.1,E2 11848.1} C_VEL
LIN {X 0,Y 476.168,Z 941.98,A -85,B 0,C 180,E1 11847.134,E2 11847.134} C_VEL
LIN {X 0,Y 469.128,Z 967.317,A -85,B 0,C 180,E1 11845.758,E2 11845.758} C_VEL
LIN {X 0,Y 462.182,Z 989.362,A -85,B 0,C 180,E1 11844.327,E2 11844.327} C_VEL
LIN {X 0,Y 455.677,Z 1008.553,A -85,B 0,C 180,E1 11842.884,E2 11842.884} C_VEL
LIN {X 0,Y 449.044,Z 1026.918,A -85,B 0,C 180,E1 11841.302,E2 11841.302} C_VEL
LIN {X 0,Y 441.498,Z 1046.726,A -85,B 0,C 180,E1 11839.349,E2 11839.349} C_VEL
LIN {X 0,Y 432.756,Z 1068.283,A -85,B 0,C 180,E1 11836.85,E2 11836.85} C_VEL
LIN {X 0,Y 425.921,Z 1084.595,A -85,B 0,C 180,E1 11834.657,E2 11834.657} C_VEL
LIN {X 0,Y 419.544,Z 1099.58,A -85,B 0,C 180,E1 11832.369,E2 11832.369} C_VEL
LIN {X 0,Y 412.71,Z 1115.583,A -85,B 0,C 180,E1 11829.582,E2 11829.582} C_VEL
LIN {X 0,Y 405.789,Z 1131.862,A -85,B 0,C 180,E1 11826.255,E2 11826.255} C_VEL
LIN {X 0,Y 400.609,Z 1144.31,A -85,B 0,C 180,E1 11823.306,E2 11823.306} C_VEL
LIN {X 0,Y 396.338,Z 1155.159,A -85,B 0,C 180,E1 11820.366,E2 11820.366} C_VEL
LIN {X 0,Y 392.537,Z 1165.573,A -85,B 0,C 180,E1 11817.127,E2 11817.127} C_VEL
LIN {X 0,Y 388.904,Z 1176.701,A -85,B 0,C 180,E1 11813.004,E2 11813.004} C_VEL
LIN {X 0,Y 386.819,Z 1184.215,A -85,B 0,C 180,E1 11809.636,E2 11809.636} C_VEL
LIN {X 0,Y 385.458,Z 1190.212,A -85,B 0,C 180,E1 11806.425,E2 11806.425} C_VEL
LIN {X 0,Y 384.633,Z 1194.887,A -85,B 0,C 180,E1 11803.378,E2 11803.378} C_VEL
LIN {X 0,Y 384.172,Z 1198.742,A -85,B 0,C 180,E1 11800.195,E2 11800.195} C_VEL
LIN {X 0,Y 383.972,Z 1201.547,A -85,B 0,C 180,E1 11797.031,E2 11797.031} C_VEL
LIN {X 0,Y 383.916,Z 1203.325,A -85,B 0,C 180,E1 11793.883,E2 11793.883} C_VEL
LIN {X 0,Y 383.903,Z 1204.134,A -85,B 0,C 180,E1 11790.448,E2 11790.448} C_VEL
LIN {X 0,Y 383.915,Z 1203.632,A -85,B 0,C 180,E1 11786.716,E2 11786.716} C_VEL
LIN {X 0,Y 383.966,Z 1201.722,A -85,B 0,C 180,E1 11783.121,E2 11783.121} C_VEL
LIN {X 0,Y 384.16,Z 1199.007,A -85,B 0,C 180,E1 11779.958,E2 11779.958} C_VEL
LIN {X 0,Y 384.607,Z 1195.267,A -85,B 0,C 180,E1 11776.776,E2 11776.776} C_VEL
LIN {X 0,Y 385.47,Z 1190.479,A -85,B 0,C 180,E1 11773.577,E2 11773.577} C_VEL
LIN {X 0,Y 386.842,Z 1184.616,A -85,B 0,C 180,E1 11770.367,E2 11770.367} C_VEL
LIN {X 0,Y 388.843,Z 1177.642,A -85,B 0,C 180,E1 11767.153,E2 11767.153} C_VEL
LIN {X 0,Y 392.172,Z 1167.896,A -85,B 0,C 180,E1 11763.339,E2 11763.339} C_VEL
LIN {X 0,Y 396.622,Z 1156.21,A -85,B 0,C 180,E1 11759.555,E2 11759.555} C_VEL
LIN {X 0,Y 401.33,Z 1144.955,A -85,B 0,C 180,E1 11756.421,E2 11756.421} C_VEL
LIN {X 0,Y 406.606,Z 1133.06,A -85,B 0,C 180,E1 11753.527,E2 11753.527} C_VEL
LIN {X 0,Y 413.843,Z 1117.316,A -85,B 0,C 180,E1 11750.19,E2 11750.19} C_VEL
LIN {X 0,Y 421.836,Z 1099.909,A -85,B 0,C 180,E1 11747.091,E2 11747.091} C_VEL
LIN {X 0,Y 428.69,Z 1085.023,A -85,B 0,C 180,E1 11744.781,E2 11744.781} C_VEL
LIN {X 0,Y 435.971,Z 1068.969,A -85,B 0,C 180,E1 11742.593,E2 11742.593} C_VEL
LIN {X 0,Y 445.177,Z 1048.158,A -85,B 0,C 180,E1 11740.137,E2 11740.137} C_VEL
LIN {X 0,Y 453.834,Z 1027.184,A -85,B 0,C 180,E1 11738.053,E2 11738.053} C_VEL
LIN {X 0,Y 460.889,Z 1009.174,A -85,B 0,C 180,E1 11736.498,E2 11736.498} C_VEL
LIN {X 0,Y 467.874,Z 990.199,A -85,B 0,C 180,E1 11735.067,E2 11735.067} C_VEL
LIN {X 0,Y 475.199,Z 968.811,A -85,B 0,C 180,E1 11733.678,E2 11733.678} C_VEL
LIN {X 0,Y 483.204,Z 942.507,A -85,B 0,C 180,E1 11732.25,E2 11732.25} C_VEL
LIN {X 0,Y 489.008,Z 920.884,A -85,B 0,C 180,E1 11731.276,E2 11731.276} C_VEL
LIN {X 0,Y 493.814,Z 900.677,A -85,B 0,C 180,E1 11730.51,E2 11730.51} C_VEL
LIN {X 0,Y 498.145,Z 879.62,A -85,B 0,C 180,E1 11729.841,E2 11729.841} C_VEL
LIN {X 0,Y 502.322,Z 855.451,A -85,B 0,C 180,E1 11729.226,E2 11729.226} C_VEL
LIN {X 0,Y 505.942,Z 826.436,A -85,B 0,C 180,E1 11728.664,E2 11728.664} C_VEL
LIN {X 0,Y 511.235,Z 754.503,A -85,B 0,C 180,E1 11727.523,E2 11727.523} C_VEL
LIN {X 0,Y 527.225,Z 535.368,A -85,B 0,C 180,E1 11724.109,E2 11724.109} C_VEL
LIN {X 0,Y 528.063,Z 523.403,A -85,B 0,C 180,E1 11723.904,E2 11723.904} C_VEL
LIN {X 0,Y 519.77,Z 509.573,A -85,B 0,C 180,E1 11720.848,E2 11720.848} C_VEL
LIN {X 0,Y 514.954,Z 502.467,A -85,B 0,C 180,E1 11718.804,E2 11718.804} C_VEL
LIN {X 0,Y 511.539,Z 497.634,A -85,B 0,C 180,E1 11717.167,E2 11717.167} C_VEL
LIN {X 0,Y 508.308,Z 493.041,A -85,B 0,C 180,E1 11715.4,E2 11715.4} C_VEL
LIN {X 0,Y 504.859,Z 488.233,A -85,B 0,C 180,E1 11713.165,E2 11713.165} C_VEL
LIN {X 0,Y 501.965,Z 484.254,A -85,B 0,C 180,E1 11710.792,E2 11710.792} C_VEL
LIN {X 0,Y 501.312,Z 483.018,A -85,B 0,C 180,E1 11710.109,E2 11710.109} C_VEL
LIN {X 0,Y 498.273,Z 479.286,A -85,B 0,C 180,E1 11705.527,E2 11705.527} C_VEL
LIN {X 0,Y 497.991,Z 477.263,A -85,B 0,C 180,E1 11703.223,E2 11703.223} C_VEL
LIN {X 0,Y 498.003,Z 477.551,A -85,B 0,C 180,E1 11702.071,E2 11702.071} C_VEL
LIN {X 0,Y 500.67,Z 482.555,A -85,B 0,C 180,E1 11696.336,E2 11696.336} C_VEL
LIN {X 0,Y 501.614,Z 483.516,A -85,B 0,C 180,E1 11695.369,E2 11695.369} C_VEL
LIN {X 0,Y 504.578,Z 487.924,A -85,B 0,C 180,E1 11692.828,E2 11692.828} C_VEL
LIN {X 0,Y 505.697,Z 489.37,A -85,B 0,C 180,E1 11692.044,E2 11692.044} C_VEL
LIN {X 0,Y 509.615,Z 494.764,A -85,B 0,C 180,E1 11689.658,E2 11689.658} C_VEL
LIN {X 0,Y 513.46,Z 500.275,A -85,B 0,C 180,E1 11687.688,E2 11687.688} C_VEL
LIN {X 0,Y 517.953,Z 506.725,A -85,B 0,C 180,E1 11685.694,E2 11685.694} C_VEL
LIN {X 0,Y 523.681,Z 515.209,A -85,B 0,C 180,E1 11683.471,E2 11683.471} C_VEL
LIN {X 0,Y 528.092,Z 522.099,A -85,B 0,C 180,E1 11681.931,E2 11681.931} C_VEL
LIN {X 0,Y 512.843,Z 729.738,A -85,B 0,C 180,E1 11678.695,E2 11678.695} C_VEL
LIN {X 0,Y 506.215,Z 820.553,A -85,B 0,C 180,E1 11677.261,E2 11677.261} C_VEL
LIN {X 0,Y 502.862,Z 848.423,A -85,B 0,C 180,E1 11676.725,E2 11676.725} C_VEL
LIN {X 0,Y 498.542,Z 873.855,A -85,B 0,C 180,E1 11676.07,E2 11676.07} C_VEL
LIN {X 0,Y 494.257,Z 894.862,A -85,B 0,C 180,E1 11675.398,E2 11675.398} C_VEL
LIN {X 0,Y 489.445,Z 915.266,A -85,B 0,C 180,E1 11674.616,E2 11674.616} C_VEL
LIN {X 0,Y 483.877,Z 936.145,A -85,B 0,C 180,E1 11673.667,E2 11673.667} C_VEL
LIN {X 0,Y 476.439,Z 960.978,A -85,B 0,C 180,E1 11672.327,E2 11672.327} C_VEL
LIN {X 0,Y 468.739,Z 983.496,A -85,B 0,C 180,E1 11670.868,E2 11670.868} C_VEL
LIN {X 0,Y 461.95,Z 1001.943,A -85,B 0,C 180,E1 11669.479,E2 11669.479} C_VEL
LIN {X 0,Y 454.883,Z 1019.975,A -85,B 0,C 180,E1 11667.925,E2 11667.925} C_VEL
LIN {X 0,Y 447.344,Z 1038.151,A -85,B 0,C 180,E1 11666.134,E2 11666.134} C_VEL
LIN {X 0,Y 437.744,Z 1060.058,A -85,B 0,C 180,E1 11663.614,E2 11663.614} C_VEL
LIN {X 0,Y 429.736,Z 1077.489,A -85,B 0,C 180,E1 11661.252,E2 11661.252} C_VEL
LIN {X 0,Y 422.851,Z 1092.241,A -85,B 0,C 180,E1 11658.964,E2 11658.964} C_VEL
LIN {X 0,Y 415.918,Z 1107.014,A -85,B 0,C 180,E1 11656.352,E2 11656.352} C_VEL
LIN {X 0,Y 407.854,Z 1124.318,A -85,B 0,C 180,E1 11652.771,E2 11652.771} C_VEL
LIN {X 0,Y 402.122,Z 1136.868,A -85,B 0,C 180,E1 11649.719,E2 11649.719} C_VEL
LIN {X 0,Y 397.542,Z 1147.452,A -85,B 0,C 180,E1 11646.769,E2 11646.769} C_VEL
LIN {X 0,Y 393.403,Z 1157.746,A -85,B 0,C 180,E1 11643.471,E2 11643.471} C_VEL
LIN {X 0,Y 389.364,Z 1168.973,A -85,B 0,C 180,E1 11639.176,E2 11639.176} C_VEL
LIN {X 0,Y 387.078,Z 1176.417,A -85,B 0,C 180,E1 11635.719,E2 11635.719} C_VEL
LIN {X 0,Y 385.664,Z 1182.113,A -85,B 0,C 180,E1 11632.563,E2 11632.563} C_VEL
LIN {X 0,Y 384.722,Z 1186.854,A -85,B 0,C 180,E1 11629.363,E2 11629.363} C_VEL
LIN {X 0,Y 384.232,Z 1190.531,A -85,B 0,C 180,E1 11626.207,E2 11626.207} C_VEL
LIN {X 0,Y 383.999,Z 1193.202,A -85,B 0,C 180,E1 11623.093,E2 11623.093} C_VEL
LIN {X 0,Y 383.924,Z 1195.024,A -85,B 0,C 180,E1 11619.746,E2 11619.746} C_VEL
LIN {X 0,Y 383.91,Z 1195.801,A -85,B 0,C 180,E1 11615.979,E2 11615.979} C_VEL
LIN {X 0,Y 383.924,Z 1195.011,A -85,B 0,C 180,E1 11612.238,E2 11612.238} C_VEL
LIN {X 0,Y 383.993,Z 1193.216,A -85,B 0,C 180,E1 11608.955,E2 11608.955} C_VEL
LIN {X 0,Y 384.205,Z 1190.509,A -85,B 0,C 180,E1 11605.821,E2 11605.821} C_VEL
LIN {X 0,Y 384.694,Z 1186.808,A -85,B 0,C 180,E1 11602.682,E2 11602.682} C_VEL
LIN {X 0,Y 385.467,Z 1182.576,A -85,B 0,C 180,E1 11599.831,E2 11599.831} C_VEL
LIN {X 0,Y 384.879,Z 1180.797,A -85,B 0,C 180,E1 11598.71,E2 11598.71} C_VEL
LIN {X 0,Y 380.022,Z 1175.735,A -85,B 0,C 180,E1 11595.611,E2 11595.611} C_VEL
LIN {X 0,Y 379.888,Z 1173.918,A -85,B 0,C 180,E1 11594.729,E2 11594.729} C_VEL
LIN {X 0,Y 382.87,Z 1164.636,A -85,B 0,C 180,E1 11590.788,E2 11590.788} C_VEL
LIN {X 0,Y 386.108,Z 1155.875,A -85,B 0,C 180,E1 11587.624,E2 11587.624} C_VEL
LIN {X 0,Y 389.908,Z 1146.371,A -85,B 0,C 180,E1 11584.643,E2 11584.643} C_VEL
LIN {X 0,Y 394.897,Z 1134.766,A -85,B 0,C 180,E1 11581.476,E2 11581.476} C_VEL
LIN {X 0,Y 402.028,Z 1118.628,A -85,B 0,C 180,E1 11577.739,E2 11577.739} C_VEL
LIN {X 0,Y 408.227,Z 1104.92,A -85,B 0,C 180,E1 11575.03,E2 11575.03} C_VEL
LIN {X 0,Y 414.248,Z 1091.589,A -85,B 0,C 180,E1 11572.71,E2 11572.71} C_VEL
LIN {X 0,Y 420.806,Z 1076.875,A -85,B 0,C 180,E1 11570.446,E2 11570.446} C_VEL
LIN {X 0,Y 429.264,Z 1057.628,A -85,B 0,C 180,E1 11567.868,E2 11567.868} C_VEL
LIN {X 0,Y 437.69,Z 1037.191,A -85,B 0,C 180,E1 11565.558,E2 11565.558} C_VEL
LIN {X 0,Y 444.488,Z 1019.918,A -85,B 0,C 180,E1 11563.857,E2 11563.857} C_VEL
LIN {X 0,Y 451.314,Z 1001.55,A -85,B 0,C 180,E1 11562.271,E2 11562.271} C_VEL
LIN {X 0,Y 458.51,Z 980.862,A -85,B 0,C 180,E1 11560.72,E2 11560.72} C_VEL
LIN {X 0,Y 466.499,Z 955.429,A -85,B 0,C 180,E1 11559.113,E2 11559.113} C_VEL
LIN {X 0,Y 472.452,Z 934.149,A -85,B 0,C 180,E1 11557.984,E2 11557.984} C_VEL
LIN {X 0,Y 477.642,Z 913.43,A -85,B 0,C 180,E1 11557.047,E2 11557.047} C_VEL
LIN {X 0,Y 482.42,Z 891.732,A -85,B 0,C 180,E1 11556.219,E2 11556.219} C_VEL
LIN {X 0,Y 487.476,Z 864.34,A -85,B 0,C 180,E1 11555.374,E2 11555.374} C_VEL
LIN {X 0,Y 491.031,Z 839.332,A -85,B 0,C 180,E1 11554.789,E2 11554.789} C_VEL
LIN {X 0,Y 493.368,Z 816.959,A -85,B 0,C 180,E1 11554.376,E2 11554.376} C_VEL
LIN {X 0,Y 507.492,Z 602.689,A -85,B 0,C 180,E1 11551.026,E2 11551.026} C_VEL
LIN {X 0,Y 512.95,Z 521.098,A -85,B 0,C 180,E1 11549.742,E2 11549.742} C_VEL
LIN {X 0,Y 503.732,Z 506.926,A -85,B 0,C 180,E1 11547.037,E2 11547.037} C_VEL
LIN {X 0,Y 494.811,Z 493.827,A -85,B 0,C 180,E1 11544.024,E2 11544.024} C_VEL
LIN {X 0,Y 487.69,Z 483.883,A -85,B 0,C 180,E1 11541.215,E2 11541.215} C_VEL
LIN {X 0,Y 483.514,Z 478.343,A -85,B 0,C 180,E1 11539.322,E2 11539.322} C_VEL
LIN {X 0,Y 479.905,Z 473.477,A -85,B 0,C 180,E1 11537.459,E2 11537.459} C_VEL
LIN {X 0,Y 476.188,Z 468.469,A -85,B 0,C 180,E1 11535.217,E2 11535.217} C_VEL
LIN {X 0,Y 472.923,Z 464.352,A -85,B 0,C 180,E1 11532.827,E2 11532.827} C_VEL
LIN {X 0,Y 472.124,Z 462.926,A -85,B 0,C 180,E1 11532.103,E2 11532.103} C_VEL
LIN {X 0,Y 469.24,Z 459.989,A -85,B 0,C 180,E1 11529.073,E2 11529.073} C_VEL
LIN {X 0,Y 468.122,Z 457.178,A -85,B 0,C 180,E1 11526.993,E2 11526.993} C_VEL
LIN {X 0,Y 467.368,Z 456.908,A -85,B 0,C 180,E1 11520.981,E2 11520.981} C_VEL
LIN {X 0,Y 468.279,Z 457.478,A -85,B 0,C 180,E1 11518.777,E2 11518.777} C_VEL
LIN {X 0,Y 469.963,Z 461.121,A -85,B 0,C 180,E1 11516.096,E2 11516.096} C_VEL
LIN {X 0,Y 472.543,Z 463.592,A -85,B 0,C 180,E1 11513.622,E2 11513.622} C_VEL
LIN {X 0,Y 475.55,Z 467.962,A -85,B 0,C 180,E1 11511.293,E2 11511.293} C_VEL
LIN {X 0,Y 476.925,Z 469.51,A -85,B 0,C 180,E1 11510.405,E2 11510.405} C_VEL
LIN {X 0,Y 480.982,Z 474.915,A -85,B 0,C 180,E1 11508.062,E2 11508.062} C_VEL
LIN {X 0,Y 485.565,Z 481.217,A -85,B 0,C 180,E1 11505.815,E2 11505.815} C_VEL
LIN {X 0,Y 489.375,Z 486.441,A -85,B 0,C 180,E1 11504.171,E2 11504.171} C_VEL
LIN {X 0,Y 495.707,Z 495.227,A -85,B 0,C 180,E1 11501.75,E2 11501.75} C_VEL
LIN {X 0,Y 502.448,Z 505.205,A -85,B 0,C 180,E1 11499.467,E2 11499.467} C_VEL
LIN {X 0,Y 512.161,Z 521.49,A -85,B 0,C 180,E1 11496.53,E2 11496.53} C_VEL
LIN {X 0,Y 512.977,Z 523.147,A -85,B 0,C 180,E1 11496.292,E2 11496.292} C_VEL
LIN {X 0,Y 498.599,Z 739.987,A -85,B 0,C 180,E1 11492.914,E2 11492.914} C_VEL
LIN {X 0,Y 492.888,Z 825.792,A -85,B 0,C 180,E1 11491.559,E2 11491.559} C_VEL
LIN {X 0,Y 489.707,Z 853.726,A -85,B 0,C 180,E1 11491.019,E2 11491.019} C_VEL
LIN {X 0,Y 485.537,Z 879.348,A -85,B 0,C 180,E1 11490.361,E2 11490.361} C_VEL
LIN {X 0,Y 481.382,Z 900.743,A -85,B 0,C 180,E1 11489.671,E2 11489.671} C_VEL
LIN {X 0,Y 476.792,Z 921.14,A -85,B 0,C 180,E1 11488.886,E2 11488.886} C_VEL
LIN {X 0,Y 471.129,Z 943.435,A -85,B 0,C 180,E1 11487.866,E2 11487.866} C_VEL
LIN {X 0,Y 463.417,Z 970.046,A -85,B 0,C 180,E1 11486.392,E2 11486.392} C_VEL
LIN {X 0,Y 456.765,Z 990.522,A -85,B 0,C 180,E1 11485.047,E2 11485.047} C_VEL
LIN {X 0,Y 450.256,Z 1009.163,A -85,B 0,C 180,E1 11483.635,E2 11483.635} C_VEL
LIN {X 0,Y 443.082,Z 1028.438,A -85,B 0,C 180,E1 11481.959,E2 11481.959} C_VEL
LIN {X 0,Y 434.094,Z 1051.068,A -85,B 0,C 180,E1 11479.665,E2 11479.665} C_VEL
LIN {X 0,Y 426.246,Z 1069.689,A -85,B 0,C 180,E1 11477.441,E2 11477.441} C_VEL
LIN {X 0,Y 419.378,Z 1085.537,A -85,B 0,C 180,E1 11475.275,E2 11475.275} C_VEL
LIN {X 0,Y 412.669,Z 1100.748,A -85,B 0,C 180,E1 11472.911,E2 11472.911} C_VEL
LIN {X 0,Y 404.893,Z 1118.3,A -85,B 0,C 180,E1 11469.762,E2 11469.762} C_VEL
LIN {X 0,Y 398.423,Z 1132.881,A -85,B 0,C 180,E1 11466.676,E2 11466.676} C_VEL
LIN {X 0,Y 393.191,Z 1144.989,A -85,B 0,C 180,E1 11463.74,E2 11463.74} C_VEL
LIN {X 0,Y 388.806,Z 1155.652,A -85,B 0,C 180,E1 11460.782,E2 11460.782} C_VEL
LIN {X 0,Y 384.285,Z 1167.67,A -85,B 0,C 180,E1 11456.92,E2 11456.92} C_VEL
LIN {X 0,Y 380.901,Z 1177.604,A -85,B 0,C 180,E1 11453.025,E2 11453.025} C_VEL
LIN {X 0,Y 378.948,Z 1184.365,A -85,B 0,C 180,E1 11449.9,E2 11449.9} C_VEL
LIN {X 0,Y 377.569,Z 1190.069,A -85,B 0,C 180,E1 11446.778,E2 11446.778} C_VEL
LIN {X 0,Y 376.698,Z 1194.757,A -85,B 0,C 180,E1 11443.665,E2 11443.665} C_VEL
LIN {X 0,Y 376.209,Z 1198.461,A -85,B 0,C 180,E1 11440.568,E2 11440.568} C_VEL
LIN {X 0,Y 375.999,Z 1201.209,A -85,B 0,C 180,E1 11437.488,E2 11437.488} C_VEL
LIN {X 0,Y 375.919,Z 1203.019,A -85,B 0,C 180,E1 11434.424,E2 11434.424} C_VEL
LIN {X 0,Y 375.914,Z 1203.884,A -85,B 0,C 180,E1 11431.525,E2 11431.525} C_VEL
LIN {X 0,Y 375.915,Z 1203.924,A -85,B 0,C 180,E1 11428.629,E2 11428.629} C_VEL
LIN {X 0,Y 375.918,Z 1203.073,A -85,B 0,C 180,E1 11425.577,E2 11425.577} C_VEL
LIN {X 0,Y 375.998,Z 1201.309,A -85,B 0,C 180,E1 11422.513,E2 11422.513} C_VEL
LIN {X 0,Y 376.211,Z 1198.626,A -85,B 0,C 180,E1 11419.434,E2 11419.434} C_VEL
LIN {X 0,Y 376.741,Z 1194.803,A -85,B 0,C 180,E1 11416.181,E2 11416.181} C_VEL
LIN {X 0,Y 377.639,Z 1190.188,A -85,B 0,C 180,E1 11413.068,E2 11413.068} C_VEL
LIN {X 0,Y 379.154,Z 1184.291,A -85,B 0,C 180,E1 11409.791,E2 11409.791} C_VEL
LIN {X 0,Y 381.55,Z 1176.577,A -85,B 0,C 180,E1 11406.199,E2 11406.199} C_VEL
LIN {X 0,Y 385.817,Z 1165.03,A -85,B 0,C 180,E1 11401.782,E2 11401.782} C_VEL
LIN {X 0,Y 390.068,Z 1154.719,A -85,B 0,C 180,E1 11398.472,E2 11398.472} C_VEL
LIN {X 0,Y 394.904,Z 1143.886,A -85,B 0,C 180,E1 11395.449,E2 11395.449} C_VEL
LIN {X 0,Y 400.863,Z 1131.097,A -85,B 0,C 180,E1 11392.331,E2 11392.331} C_VEL
LIN {X 0,Y 409.23,Z 1113.653,A -85,B 0,C 180,E1 11388.724,E2 11388.724} C_VEL
LIN {X 0,Y 416.072,Z 1099.445,A -85,B 0,C 180,E1 11386.204,E2 11386.204} C_VEL
LIN {X 0,Y 423.174,Z 1084.607,A -85,B 0,C 180,E1 11383.892,E2 11383.892} C_VEL
LIN {X 0,Y 430.634,Z 1068.743,A -85,B 0,C 180,E1 11381.723,E2 11381.723} C_VEL
LIN {X 0,Y 439.953,Z 1048.378,A -85,B 0,C 180,E1 11379.309,E2 11379.309} C_VEL
LIN {X 0,Y 448.883,Z 1027.418,A -85,B 0,C 180,E1 11377.221,E2 11377.221} C_VEL
LIN {X 0,Y 456.122,Z 1009.5,A -85,B 0,C 180,E1 11375.67,E2 11375.67} C_VEL
LIN {X 0,Y 463.262,Z 990.645,A -85,B 0,C 180,E1 11374.246,E2 11374.246} C_VEL
LIN {X 0,Y 470.464,Z 970.208,A -85,B 0,C 180,E1 11372.915,E2 11372.915} C_VEL
LIN {X 0,Y 478.778,Z 943.89,A -85,B 0,C 180,E1 11371.474,E2 11371.474} C_VEL
LIN {X 0,Y 484.913,Z 921.658,A -85,B 0,C 180,E1 11370.47,E2 11370.47} C_VEL
LIN {X 0,Y 489.989,Z 900.852,A -85,B 0,C 180,E1 11369.683,E2 11369.683} C_VEL
LIN {X 0,Y 494.479,Z 879.527,A -85,B 0,C 180,E1 11369.01,E2 11369.01} C_VEL
LIN {X 0,Y 498.747,Z 855.364,A -85,B 0,C 180,E1 11368.4,E2 11368.4} C_VEL
LIN {X 0,Y 502.443,Z 826.371,A -85,B 0,C 180,E1 11367.841,E2 11367.841} C_VEL
LIN {X 0,Y 507.808,Z 755.434,A -85,B 0,C 180,E1 11366.717,E2 11366.717} C_VEL
LIN {X 0,Y 524.23,Z 536.428,A -85,B 0,C 180,E1 11363.308,E2 11363.308} C_VEL
LIN {X 0,Y 524.78,Z 528.587,A -85,B 0,C 180,E1 11363.17,E2 11363.17} C_VEL
LIN {X 0,Y 517.659,Z 516.447,A -85,B 0,C 180,E1 11360.434,E2 11360.434} C_VEL
LIN {X 0,Y 513.26,Z 509.866,A -85,B 0,C 180,E1 11358.514,E2 11358.514} C_VEL
LIN {X 0,Y 509.919,Z 505.061,A -85,B 0,C 180,E1 11356.871,E2 11356.871} C_VEL
LIN {X 0,Y 506.956,Z 500.744,A -85,B 0,C 180,E1 11355.208,E2 11355.208} C_VEL
LIN {X 0,Y 503.733,Z 496.118,A -85,B 0,C 180,E1 11353.079,E2 11353.079} C_VEL
LIN {X 0,Y 500.812,Z 492.073,A -85,B 0,C 180,E1 11350.643,E2 11350.643} C_VEL
LIN {X 0,Y 500.112,Z 490.841,A -85,B 0,C 180,E1 11349.901,E2 11349.901} C_VEL
LIN {X 0,Y 497.202,Z 486.958,A -85,B 0,C 180,E1 11345.192,E2 11345.192} C_VEL
LIN {X 0,Y 497.009,Z 485.206,A -85,B 0,C 180,E1 11343.114,E2 11343.114} C_VEL
LIN {X 0,Y 497.021,Z 485.53,A -85,B 0,C 180,E1 11342.075,E2 11342.075} C_VEL
LIN {X 0,Y 499.587,Z 490.438,A -85,B 0,C 180,E1 11336.443,E2 11336.443} C_VEL
LIN {X 0,Y 500.46,Z 491.314,A -85,B 0,C 180,E1 11335.531,E2 11335.531} C_VEL
LIN {X 0,Y 503.439,Z 495.797,A -85,B 0,C 180,E1 11332.927,E2 11332.927} C_VEL
LIN {X 0,Y 504.535,Z 497.332,A -85,B 0,C 180,E1 11332.14,E2 11332.14} C_VEL
LIN {X 0,Y 508.221,Z 502.45,A -85,B 0,C 180,E1 11329.858,E2 11329.858} C_VEL
LIN {X 0,Y 512.002,Z 507.977,A -85,B 0,C 180,E1 11327.881,E2 11327.881} C_VEL
LIN {X 0,Y 517.475,Z 515.826,A -85,B 0,C 180,E1 11325.452,E2 11325.452} C_VEL
LIN {X 0,Y 524.405,Z 526.613,A -85,B 0,C 180,E1 11322.81,E2 11322.81} C_VEL
LIN {X 0,Y 524.791,Z 527.489,A -85,B 0,C 180,E1 11322.664,E2 11322.664} C_VEL
LIN {X 0,Y 509.255,Z 733.606,A -85,B 0,C 180,E1 11319.456,E2 11319.456} C_VEL
LIN {X 0,Y 502.712,Z 820.739,A -85,B 0,C 180,E1 11318.08,E2 11318.08} C_VEL
LIN {X 0,Y 499.265,Z 848.69,A -85,B 0,C 180,E1 11317.543,E2 11317.543} C_VEL
LIN {X 0,Y 494.855,Z 874.059,A -85,B 0,C 180,E1 11316.895,E2 11316.895} C_VEL
LIN {X 0,Y 490.532,Z 894.806,A -85,B 0,C 180,E1 11316.235,E2 11316.235} C_VEL
LIN {X 0,Y 485.576,Z 915.358,A -85,B 0,C 180,E1 11315.453,E2 11315.453} C_VEL
LIN {X 0,Y 480.058,Z 935.592,A -85,B 0,C 180,E1 11314.541,E2 11314.541} C_VEL
LIN {X 0,Y 472.572,Z 960.113,A -85,B 0,C 180,E1 11313.235,E2 11313.235} C_VEL
LIN {X 0,Y 464.347,Z 983.576,A -85,B 0,C 180,E1 11311.723,E2 11311.723} C_VEL
LIN {X 0,Y 457.085,Z 1002.764,A -85,B 0,C 180,E1 11310.277,E2 11310.277} C_VEL
LIN {X 0,Y 449.825,Z 1020.717,A -85,B 0,C 180,E1 11308.722,E2 11308.722} C_VEL
LIN {X 0,Y 441.8,Z 1039.454,A -85,B 0,C 180,E1 11306.863,E2 11306.863} C_VEL
LIN {X 0,Y 431.791,Z 1061.413,A -85,B 0,C 180,E1 11304.299,E2 11304.299} C_VEL
LIN {X 0,Y 424.077,Z 1077.644,A -85,B 0,C 180,E1 11302.079,E2 11302.079} C_VEL
LIN {X 0,Y 417.145,Z 1091.945,A -85,B 0,C 180,E1 11299.85,E2 11299.85} C_VEL
LIN {X 0,Y 410.223,Z 1106.081,A -85,B 0,C 180,E1 11297.343,E2 11297.343} C_VEL
LIN {X 0,Y 402.459,Z 1122.08,A -85,B 0,C 180,E1 11294.077,E2 11294.077} C_VEL
LIN {X 0,Y 395.739,Z 1136.032,A -85,B 0,C 180,E1 11290.681,E2 11290.681} C_VEL
LIN {X 0,Y 390.834,Z 1146.705,A -85,B 0,C 180,E1 11287.693,E2 11287.693} C_VEL
LIN {X 0,Y 386.559,Z 1156.62,A -85,B 0,C 180,E1 11284.503,E2 11284.503} C_VEL
LIN {X 0,Y 382.717,Z 1166.51,A -85,B 0,C 180,E1 11280.801,E2 11280.801} C_VEL
LIN {X 0,Y 379.593,Z 1175.7,A -85,B 0,C 180,E1 11276.601,E2 11276.601} C_VEL
LIN {X 0,Y 377.915,Z 1181.783,A -85,B 0,C 180,E1 11273.217,E2 11273.217} C_VEL
LIN {X 0,Y 376.891,Z 1186.514,A -85,B 0,C 180,E1 11270.012,E2 11270.012} C_VEL
LIN {X 0,Y 376.314,Z 1190.237,A -85,B 0,C 180,E1 11266.834,E2 11266.834} C_VEL
LIN {X 0,Y 376.032,Z 1192.989,A -85,B 0,C 180,E1 11263.688,E2 11263.688} C_VEL
LIN {X 0,Y 375.934,Z 1194.728,A -85,B 0,C 180,E1 11260.729,E2 11260.729} C_VEL
LIN {X 0,Y 375.917,Z 1195.635,A -85,B 0,C 180,E1 11257.796,E2 11257.796} C_VEL
LIN {X 0,Y 375.907,Z 1195.702,A -85,B 0,C 180,E1 11254.729,E2 11254.729} C_VEL
LIN {X 0,Y 375.929,Z 1194.873,A -85,B 0,C 180,E1 11251.676,E2 11251.676} C_VEL
LIN {X 0,Y 376.009,Z 1193.153,A -85,B 0,C 180,E1 11248.628,E2 11248.628} C_VEL
LIN {X 0,Y 376.235,Z 1190.541,A -85,B 0,C 180,E1 11245.579,E2 11245.579} C_VEL
LIN {X 0,Y 376.766,Z 1186.823,A -85,B 0,C 180,E1 11242.374,E2 11242.374} C_VEL
LIN {X 0,Y 377.694,Z 1182.092,A -85,B 0,C 180,E1 11239.166,E2 11239.166} C_VEL
LIN {X 0,Y 379.171,Z 1176.317,A -85,B 0,C 180,E1 11235.959,E2 11235.959} C_VEL
LIN {X 0,Y 379.888,Z 1173.918,A -85,B 0,C 180,E1 11234.729,E2 11234.729} C_VEL
LIN {X 0,Y 379.604,Z 1171.566,A -85,B 0,C 180,E1 11233.615,E2 11233.615} C_VEL
LIN {X 0,Y 375.776,Z 1165.366,A -85,B 0,C 180,E1 11230.584,E2 11230.584} C_VEL
LIN {X 0,Y 375.93,Z 1163.033,A -85,B 0,C 180,E1 11229.629,E2 11229.629} C_VEL
LIN {X 0,Y 379.918,Z 1153.096,A -85,B 0,C 180,E1 11226.089,E2 11226.089} C_VEL
LIN {X 0,Y 385.592,Z 1139.926,A -85,B 0,C 180,E1 11222.161,E2 11222.161} C_VEL
LIN {X 0,Y 391.129,Z 1127.782,A -85,B 0,C 180,E1 11219.08,E2 11219.08} C_VEL
LIN {X 0,Y 396.577,Z 1116.111,A -85,B 0,C 180,E1 11216.484,E2 11216.484} C_VEL
LIN {X 0,Y 403.016,Z 1102.424,A -85,B 0,C 180,E1 11213.809,E2 11213.809} C_VEL
LIN {X 0,Y 411.365,Z 1084.668,A -85,B 0,C 180,E1 11210.804,E2 11210.804} C_VEL
LIN {X 0,Y 419.714,Z 1066.151,A -85,B 0,C 180,E1 11208.161,E2 11208.161} C_VEL
LIN {X 0,Y 426.966,Z 1049.677,A -85,B 0,C 180,E1 11206.117,E2 11206.117} C_VEL
LIN {X 0,Y 434.265,Z 1032.387,A -85,B 0,C 180,E1 11204.239,E2 11204.239} C_VEL
LIN {X 0,Y 443.108,Z 1010.256,A -85,B 0,C 180,E1 11202.16,E2 11202.16} C_VEL
LIN {X 0,Y 451.135,Z 988.174,A -85,B 0,C 180,E1 11200.419,E2 11200.419} C_VEL
LIN {X 0,Y 457.548,Z 969.153,A -85,B 0,C 180,E1 11199.124,E2 11199.124} C_VEL
LIN {X 0,Y 463.554,Z 949.652,A -85,B 0,C 180,E1 11197.965,E2 11197.965} C_VEL
LIN {X 0,Y 469.763,Z 927.463,A -85,B 0,C 180,E1 11196.84,E2 11196.84} C_VEL
LIN {X 0,Y 476.426,Z 899.747,A -85,B 0,C 180,E1 11195.688,E2 11195.688} C_VEL
LIN {X 0,Y 480.933,Z 877.48,A -85,B 0,C 180,E1 11194.942,E2 11194.942} C_VEL
LIN {X 0,Y 484.53,Z 856.282,A -85,B 0,C 180,E1 11194.36,E2 11194.36} C_VEL
LIN {X 0,Y 487.612,Z 833.841,A -85,B 0,C 180,E1 11193.872,E2 11193.872} C_VEL
LIN {X 0,Y 490.348,Z 803.877,A -85,B 0,C 180,E1 11193.352,E2 11193.352} C_VEL
LIN {X 0,Y 505.348,Z 580.785,A -85,B 0,C 180,E1 11189.875,E2 11189.875} C_VEL
LIN {X 0,Y 509.065,Z 525.773,A -85,B 0,C 180,E1 11188.99,E2 11188.99} C_VEL
LIN {X 0,Y 500.621,Z 512.729,A -85,B 0,C 180,E1 11186.417,E2 11186.417} C_VEL
LIN {X 0,Y 492.632,Z 500.835,A -85,B 0,C 180,E1 11183.632,E2 11183.632} C_VEL
LIN {X 0,Y 486.058,Z 491.442,A -85,B 0,C 180,E1 11180.974,E2 11180.974} C_VEL
LIN {X 0,Y 481.828,Z 485.766,A -85,B 0,C 180,E1 11179.015,E2 11179.015} C_VEL
LIN {X 0,Y 478.404,Z 481.069,A -85,B 0,C 180,E1 11177.202,E2 11177.202} C_VEL
LIN {X 0,Y 474.857,Z 476.198,A -85,B 0,C 180,E1 11175.011,E2 11175.011} C_VEL
LIN {X 0,Y 471.666,Z 472.053,A -85,B 0,C 180,E1 11172.612,E2 11172.612} C_VEL
LIN {X 0,Y 470.878,Z 470.721,A -85,B 0,C 180,E1 11171.887,E2 11171.887} C_VEL
LIN {X 0,Y 468.096,Z 467.723,A -85,B 0,C 180,E1 11168.847,E2 11168.847} C_VEL
LIN {X 0,Y 467.088,Z 465.101,A -85,B 0,C 180,E1 11166.885,E2 11166.885} C_VEL
LIN {X 0,Y 466.426,Z 464.858,A -85,B 0,C 180,E1 11160.86,E2 11160.86} C_VEL
LIN {X 0,Y 467.236,Z 465.366,A -85,B 0,C 180,E1 11158.896,E2 11158.896} C_VEL
LIN {X 0,Y 468.878,Z 468.993,A -85,B 0,C 180,E1 11156.21,E2 11156.21} C_VEL
LIN {X 0,Y 471.346,Z 471.403,A -85,B 0,C 180,E1 11153.789,E2 11153.789} C_VEL
LIN {X 0,Y 474.391,Z 475.84,A -85,B 0,C 180,E1 11151.393,E2 11151.393} C_VEL
LIN {X 0,Y 475.652,Z 477.347,A -85,B 0,C 180,E1 11150.563,E2 11150.563} C_VEL
LIN {X 0,Y 479.547,Z 482.621,A -85,B 0,C 180,E1 11148.27,E2 11148.27} C_VEL
LIN {X 0,Y 483.941,Z 488.747,A -85,B 0,C 180,E1 11146.072,E2 11146.072} C_VEL
LIN {X 0,Y 487.96,Z 494.365,A -85,B 0,C 180,E1 11144.307,E2 11144.307} C_VEL
LIN {X 0,Y 494.232,Z 503.268,A -85,B 0,C 180,E1 11141.877,E2 11141.877} C_VEL
LIN {X 0,Y 500.335,Z 512.48,A -85,B 0,C 180,E1 11139.774,E2 11139.774} C_VEL
LIN {X 0,Y 509.167,Z 527.51,A -85,B 0,C 180,E1 11137.034,E2 11137.034} C_VEL
LIN {X 0,Y 494.363,Z 744.828,A -85,B 0,C 180,E1 11133.647,E2 11133.647} C_VEL
LIN {X 0,Y 488.786,Z 826.031,A -85,B 0,C 180,E1 11132.361,E2 11132.361} C_VEL
LIN {X 0,Y 485.458,Z 854.319,A -85,B 0,C 180,E1 11131.813,E2 11131.813} C_VEL
LIN {X 0,Y 481.256,Z 879.547,A -85,B 0,C 180,E1 11131.165,E2 11131.165} C_VEL
LIN {X 0,Y 477.121,Z 900.409,A -85,B 0,C 180,E1 11130.496,E2 11130.496} C_VEL
LIN {X 0,Y 472.427,Z 920.832,A -85,B 0,C 180,E1 11129.715,E2 11129.715} C_VEL
LIN {X 0,Y 466.781,Z 942.575,A -85,B 0,C 180,E1 11128.725,E2 11128.725} C_VEL
LIN {X 0,Y 458.87,Z 969.341,A -85,B 0,C 180,E1 11127.256,E2 11127.256} C_VEL
LIN {X 0,Y 452.089,Z 989.753,A -85,B 0,C 180,E1 11125.922,E2 11125.922} C_VEL
LIN {X 0,Y 445.361,Z 1008.58,A -85,B 0,C 180,E1 11124.499,E2 11124.499} C_VEL
LIN {X 0,Y 438.509,Z 1026.539,A -85,B 0,C 180,E1 11122.946,E2 11122.946} C_VEL
LIN {X 0,Y 431.018,Z 1045.087,A -85,B 0,C 180,E1 11121.113,E2 11121.113} C_VEL
LIN {X 0,Y 421.302,Z 1067.719,A -85,B 0,C 180,E1 11118.485,E2 11118.485} C_VEL
LIN {X 0,Y 413.919,Z 1084.205,A -85,B 0,C 180,E1 11116.243,E2 11116.243} C_VEL
LIN {X 0,Y 407.315,Z 1098.669,A -85,B 0,C 180,E1 11114.005,E2 11114.005} C_VEL
LIN {X 0,Y 400.893,Z 1112.584,A -85,B 0,C 180,E1 11111.561,E2 11111.561} C_VEL
LIN {X 0,Y 393.496,Z 1128.706,A -85,B 0,C 180,E1 11108.317,E2 11108.317} C_VEL
LIN {X 0,Y 386.891,Z 1143.217,A -85,B 0,C 180,E1 11104.831,E2 11104.831} C_VEL
LIN {X 0,Y 382.261,Z 1153.844,A -85,B 0,C 180,E1 11101.896,E2 11101.896} C_VEL
LIN {X 0,Y 378.395,Z 1163.278,A -85,B 0,C 180,E1 11098.919,E2 11098.919} C_VEL
LIN {X 0,Y 375.057,Z 1172.156,A -85,B 0,C 180,E1 11095.697,E2 11095.697} C_VEL
LIN {X 0,Y 372.028,Z 1181.378,A -85,B 0,C 180,E1 11091.771,E2 11091.771} C_VEL
LIN {X 0,Y 369.881,Z 1189.144,A -85,B 0,C 180,E1 11087.624,E2 11087.624} C_VEL
LIN {X 0,Y 368.842,Z 1194.202,A -85,B 0,C 180,E1 11084.282,E2 11084.282} C_VEL
LIN {X 0,Y 368.266,Z 1198.015,A -85,B 0,C 180,E1 11081.115,E2 11081.115} C_VEL
LIN {X 0,Y 368.013,Z 1200.867,A -85,B 0,C 180,E1 11077.965,E2 11077.965} C_VEL
LIN {X 0,Y 367.926,Z 1202.78,A -85,B 0,C 180,E1 11074.833,E2 11074.833} C_VEL
LIN {X 0,Y 367.911,Z 1203.746,A -85,B 0,C 180,E1 11071.869,E2 11071.869} C_VEL
LIN {X 0,Y 367.915,Z 1203.864,A -85,B 0,C 180,E1 11068.755,E2 11068.755} C_VEL
LIN {X 0,Y 367.918,Z 1203.068,A -85,B 0,C 180,E1 11065.637,E2 11065.637} C_VEL
LIN {X 0,Y 367.998,Z 1201.359,A -85,B 0,C 180,E1 11062.507,E2 11062.507} C_VEL
LIN {X 0,Y 368.236,Z 1198.571,A -85,B 0,C 180,E1 11059.202,E2 11059.202} C_VEL
LIN {X 0,Y 368.814,Z 1194.76,A -85,B 0,C 180,E1 11055.878,E2 11055.878} C_VEL
LIN {X 0,Y 369.795,Z 1190.077,A -85,B 0,C 180,E1 11052.647,E2 11052.647} C_VEL
LIN {X 0,Y 371.398,Z 1184.274,A -85,B 0,C 180,E1 11049.35,E2 11049.35} C_VEL
LIN {X 0,Y 373.877,Z 1176.787,A -85,B 0,C 180,E1 11045.779,E2 11045.779} C_VEL
LIN {X 0,Y 378.263,Z 1165.561,A -85,B 0,C 180,E1 11041.355,E2 11041.355} C_VEL
LIN {X 0,Y 382.722,Z 1155.288,A -85,B 0,C 180,E1 11037.972,E2 11037.972} C_VEL
LIN {X 0,Y 387.745,Z 1144.532,A -85,B 0,C 180,E1 11034.898,E2 11034.898} C_VEL
LIN {X 0,Y 393.385,Z 1132.927,A -85,B 0,C 180,E1 11031.994,E2 11031.994} C_VEL
LIN {X 0,Y 401.318,Z 1117.21,A -85,B 0,C 180,E1 11028.586,E2 11028.586} C_VEL
LIN {X 0,Y 409.681,Z 1100.457,A -85,B 0,C 180,E1 11025.537,E2 11025.537} C_VEL
LIN {X 0,Y 417.234,Z 1085.272,A -85,B 0,C 180,E1 11023.138,E2 11023.138} C_VEL
LIN {X 0,Y 424.705,Z 1069.941,A -85,B 0,C 180,E1 11021.015,E2 11021.015} C_VEL
LIN {X 0,Y 432.84,Z 1052.715,A -85,B 0,C 180,E1 11018.928,E2 11018.928} C_VEL
LIN {X 0,Y 443.153,Z 1029.745,A -85,B 0,C 180,E1 11016.56,E2 11016.56} C_VEL
LIN {X 0,Y 451.229,Z 1010.384,A -85,B 0,C 180,E1 11014.87,E2 11014.87} C_VEL
LIN {X 0,Y 458.457,Z 991.881,A -85,B 0,C 180,E1 11013.464,E2 11013.464} C_VEL
LIN {X 0,Y 465.541,Z 972.402,A -85,B 0,C 180,E1 11012.185,E2 11012.185} C_VEL
LIN {X 0,Y 472.775,Z 950.589,A -85,B 0,C 180,E1 11010.953,E2 11010.953} C_VEL
LIN {X 0,Y 480.588,Z 923.703,A -85,B 0,C 180,E1 11009.702,E2 11009.702} C_VEL
LIN {X 0,Y 485.934,Z 902.505,A -85,B 0,C 180,E1 11008.894,E2 11008.894} C_VEL
LIN {X 0,Y 490.603,Z 881.034,A -85,B 0,C 180,E1 11008.212,E2 11008.212} C_VEL
LIN {X 0,Y 494.573,Z 859.392,A -85,B 0,C 180,E1 11007.657,E2 11007.657} C_VEL
LIN {X 0,Y 498.479,Z 832.319,A -85,B 0,C 180,E1 11007.108,E2 11007.108} C_VEL
LIN {X 0,Y 502.118,Z 788.266,A -85,B 0,C 180,E1 11006.396,E2 11006.396} C_VEL
LIN {X 0,Y 519.004,Z 567.006,A -85,B 0,C 180,E1 11002.955,E2 11002.955} C_VEL
LIN {X 0,Y 521.597,Z 533.707,A -85,B 0,C 180,E1 11002.425,E2 11002.425} C_VEL
LIN {X 0,Y 515.013,Z 522.381,A -85,B 0,C 180,E1 10999.774,E2 10999.774} C_VEL
LIN {X 0,Y 511.009,Z 516.447,A -85,B 0,C 180,E1 10997.95,E2 10997.95} C_VEL
LIN {X 0,Y 508.314,Z 512.484,A -85,B 0,C 180,E1 10996.572,E2 10996.572} C_VEL
LIN {X 0,Y 505.516,Z 508.335,A -85,B 0,C 180,E1 10994.959,E2 10994.959} C_VEL
LIN {X 0,Y 502.448,Z 503.859,A -85,B 0,C 180,E1 10992.879,E2 10992.879} C_VEL
LIN {X 0,Y 499.61,Z 499.773,A -85,B 0,C 180,E1 10990.435,E2 10990.435} C_VEL
LIN {X 0,Y 498.919,Z 498.659,A -85,B 0,C 180,E1 10989.692,E2 10989.692} C_VEL
LIN {X 0,Y 496.149,Z 494.62,A -85,B 0,C 180,E1 10984.855,E2 10984.855} C_VEL
LIN {X 0,Y 496.033,Z 493.146,A -85,B 0,C 180,E1 10983.12,E2 10983.12} C_VEL
LIN {X 0,Y 496.043,Z 493.609,A -85,B 0,C 180,E1 10981.964,E2 10981.964} C_VEL
LIN {X 0,Y 498.609,Z 498.399,A -85,B 0,C 180,E1 10976.436,E2 10976.436} C_VEL
LIN {X 0,Y 499.359,Z 499.232,A -85,B 0,C 180,E1 10975.636,E2 10975.636} C_VEL
LIN {X 0,Y 502.458,Z 503.823,A -85,B 0,C 180,E1 10972.913,E2 10972.913} C_VEL
LIN {X 0,Y 506.833,Z 510.135,A -85,B 0,C 180,E1 10970.06,E2 10970.06} C_VEL
LIN {X 0,Y 510.44,Z 515.502,A -85,B 0,C 180,E1 10968.13,E2 10968.13} C_VEL
LIN {X 0,Y 515.753,Z 523.274,A -85,B 0,C 180,E1 10965.718,E2 10965.718} C_VEL
LIN {X 0,Y 521.607,Z 532.511,A -85,B 0,C 180,E1 10963.414,E2 10963.414} C_VEL
LIN {X 0,Y 505.946,Z 735.029,A -85,B 0,C 180,E1 10960.265,E2 10960.265} C_VEL
LIN {X 0,Y 499.314,Z 820.929,A -85,B 0,C 180,E1 10958.91,E2 10958.91} C_VEL
LIN {X 0,Y 495.765,Z 849.016,A -85,B 0,C 180,E1 10958.373,E2 10958.373} C_VEL
LIN {X 0,Y 491.29,Z 874.209,A -85,B 0,C 180,E1 10957.734,E2 10957.734} C_VEL
LIN {X 0,Y 486.88,Z 894.927,A -85,B 0,C 180,E1 10957.079,E2 10957.079} C_VEL
LIN {X 0,Y 481.813,Z 915.459,A -85,B 0,C 180,E1 10956.304,E2 10956.304} C_VEL
LIN {X 0,Y 475.831,Z 936.846,A -85,B 0,C 180,E1 10955.342,E2 10955.342} C_VEL
LIN {X 0,Y 467.872,Z 961.968,A -85,B 0,C 180,E1 10953.992,E2 10953.992} C_VEL
LIN {X 0,Y 459.757,Z 984.472,A -85,B 0,C 180,E1 10952.536,E2 10952.536} C_VEL
LIN {X 0,Y 452.309,Z 1003.585,A -85,B 0,C 180,E1 10951.091,E2 10951.091} C_VEL
LIN {X 0,Y 444.565,Z 1022.156,A -85,B 0,C 180,E1 10949.474,E2 10949.474} C_VEL
LIN {X 0,Y 434.95,Z 1043.794,A -85,B 0,C 180,E1 10947.284,E2 10947.284} C_VEL
LIN {X 0,Y 425.674,Z 1063.233,A -85,B 0,C 180,E1 10944.944,E2 10944.944} C_VEL
LIN {X 0,Y 418.047,Z 1078.728,A -85,B 0,C 180,E1 10942.792,E2 10942.792} C_VEL
LIN {X 0,Y 410.488,Z 1093.735,A -85,B 0,C 180,E1 10940.412,E2 10940.412} C_VEL
LIN {X 0,Y 401.73,Z 1111.009,A -85,B 0,C 180,E1 10937.241,E2 10937.241} C_VEL
LIN {X 0,Y 394.179,Z 1125.711,A -85,B 0,C 180,E1 10934.029,E2 10934.029} C_VEL
LIN {X 0,Y 388.206,Z 1137.701,A -85,B 0,C 180,E1 10931.003,E2 10931.003} C_VEL
LIN {X 0,Y 382.993,Z 1148.597,A -85,B 0,C 180,E1 10927.843,E2 10927.843} C_VEL
LIN {X 0,Y 377.707,Z 1160.577,A -85,B 0,C 180,E1 10923.773,E2 10923.773} C_VEL
LIN {X 0,Y 373.877,Z 1170.101,A -85,B 0,C 180,E1 10919.829,E2 10919.829} C_VEL
LIN {X 0,Y 371.556,Z 1176.836,A -85,B 0,C 180,E1 10916.532,E2 10916.532} C_VEL
LIN {X 0,Y 369.926,Z 1182.524,A -85,B 0,C 180,E1 10913.218,E2 10913.218} C_VEL
LIN {X 0,Y 368.887,Z 1187.1,A -85,B 0,C 180,E1 10909.969,E2 10909.969} C_VEL
LIN {X 0,Y 368.285,Z 1190.869,A -85,B 0,C 180,E1 10906.562,E2 10906.562} C_VEL
LIN {X 0,Y 367.995,Z 1193.803,A -85,B 0,C 180,E1 10902.873,E2 10902.873} C_VEL
LIN {X 0,Y 367.923,Z 1195.576,A -85,B 0,C 180,E1 10898.911,E2 10898.911} C_VEL
LIN {X 0,Y 367.905,Z 1195.85,A -85,B 0,C 180,E1 10895.145,E2 10895.145} C_VEL
LIN {X 0,Y 367.928,Z 1195.07,A -85,B 0,C 180,E1 10891.868,E2 10891.868} C_VEL
LIN {X 0,Y 368.004,Z 1193.423,A -85,B 0,C 180,E1 10888.754,E2 10888.754} C_VEL
LIN {X 0,Y 368.249,Z 1190.727,A -85,B 0,C 180,E1 10885.483,E2 10885.483} C_VEL
LIN {X 0,Y 368.808,Z 1187.037,A -85,B 0,C 180,E1 10882.209,E2 10882.209} C_VEL
LIN {X 0,Y 369.78,Z 1182.333,A -85,B 0,C 180,E1 10878.931,E2 10878.931} C_VEL
LIN {X 0,Y 371.333,Z 1176.586,A -85,B 0,C 180,E1 10875.656,E2 10875.656} C_VEL
LIN {X 0,Y 373.754,Z 1169.07,A -85,B 0,C 180,E1 10872.082,E2 10872.082} C_VEL
LIN {X 0,Y 375.93,Z 1163.033,A -85,B 0,C 180,E1 10869.629,E2 10869.629} C_VEL
LIN {X 0,Y 376.075,Z 1160.371,A -85,B 0,C 180,E1 10868.519,E2 10868.519} C_VEL
LIN {X 0,Y 373.389,Z 1153.084,A -85,B 0,C 180,E1 10865.49,E2 10865.49} C_VEL
LIN {X 0,Y 373.858,Z 1150.337,A -85,B 0,C 180,E1 10864.561,E2 10864.561} C_VEL
LIN {X 0,Y 379.306,Z 1138.416,A -85,B 0,C 180,E1 10861.068,E2 10861.068} C_VEL
LIN {X 0,Y 384.765,Z 1126.98,A -85,B 0,C 180,E1 10858.161,E2 10858.161} C_VEL
LIN {X 0,Y 390.817,Z 1114.533,A -85,B 0,C 180,E1 10855.391,E2 10855.391} C_VEL
LIN {X 0,Y 398.747,Z 1098.418,A -85,B 0,C 180,E1 10852.277,E2 10852.277} C_VEL
LIN {X 0,Y 407.436,Z 1080.168,A -85,B 0,C 180,E1 10849.317,E2 10849.317} C_VEL
LIN {X 0,Y 414.654,Z 1064.732,A -85,B 0,C 180,E1 10847.144,E2 10847.144} C_VEL
LIN {X 0,Y 422.149,Z 1048.171,A -85,B 0,C 180,E1 10845.103,E2 10845.103} C_VEL
LIN {X 0,Y 431.434,Z 1026.718,A -85,B 0,C 180,E1 10842.818,E2 10842.818} C_VEL
LIN {X 0,Y 440.171,Z 1004.642,A -85,B 0,C 180,E1 10840.849,E2 10840.849} C_VEL
LIN {X 0,Y 447.112,Z 985.906,A -85,B 0,C 180,E1 10839.408,E2 10839.408} C_VEL
LIN {X 0,Y 453.738,Z 966.619,A -85,B 0,C 180,E1 10838.121,E2 10838.121} C_VEL
LIN {X 0,Y 460.825,Z 943.866,A -85,B 0,C 180,E1 10836.808,E2 10836.808} C_VEL
LIN {X 0,Y 467.832,Z 918.048,A -85,B 0,C 180,E1 10835.587,E2 10835.587} C_VEL
LIN {X 0,Y 472.813,Z 896.929,A -85,B 0,C 180,E1 10834.757,E2 10834.757} C_VEL
LIN {X 0,Y 477.11,Z 875.851,A -85,B 0,C 180,E1 10834.066,E2 10834.066} C_VEL
LIN {X 0,Y 480.837,Z 854.011,A -85,B 0,C 180,E1 10833.48,E2 10833.48} C_VEL
LIN {X 0,Y 484.532,Z 826.341,A -85,B 0,C 180,E1 10832.906,E2 10832.906} C_VEL
LIN {X 0,Y 487.929,Z 781.317,A -85,B 0,C 180,E1 10832.178,E2 10832.178} C_VEL
LIN {X 0,Y 503.076,Z 563.206,A -85,B 0,C 180,E1 10828.777,E2 10828.777} C_VEL
LIN {X 0,Y 505.351,Z 530.634,A -85,B 0,C 180,E1 10828.255,E2 10828.255} C_VEL
LIN {X 0,Y 496.762,Z 517.239,A -85,B 0,C 180,E1 10825.515,E2 10825.515} C_VEL
LIN {X 0,Y 489.165,Z 505.976,A -85,B 0,C 180,E1 10822.727,E2 10822.727} C_VEL
LIN {X 0,Y 483.783,Z 498.204,A -85,B 0,C 180,E1 10820.444,E2 10820.444} C_VEL
LIN {X 0,Y 480.273,Z 493.33,A -85,B 0,C 180,E1 10818.763,E2 10818.763} C_VEL
LIN {X 0,Y 476.913,Z 488.658,A -85,B 0,C 180,E1 10816.943,E2 10816.943} C_VEL
LIN {X 0,Y 473.533,Z 483.925,A -85,B 0,C 180,E1 10814.803,E2 10814.803} C_VEL
LIN {X 0,Y 470.351,Z 479.622,A -85,B 0,C 180,E1 10812.336,E2 10812.336} C_VEL
LIN {X 0,Y 469.612,Z 478.495,A -85,B 0,C 180,E1 10811.645,E2 10811.645} C_VEL
LIN {X 0,Y 466.96,Z 475.455,A -85,B 0,C 180,E1 10808.621,E2 10808.621} C_VEL
LIN {X 0,Y 466.055,Z 473.024,A -85,B 0,C 180,E1 10806.777,E2 10806.777} C_VEL
LIN {X 0,Y 465.525,Z 472.821,A -85,B 0,C 180,E1 10800.615,E2 10800.615} C_VEL
LIN {X 0,Y 466.195,Z 473.254,A -85,B 0,C 180,E1 10799.017,E2 10799.017} C_VEL
LIN {X 0,Y 467.896,Z 476.986,A -85,B 0,C 180,E1 10796.202,E2 10796.202} C_VEL
LIN {X 0,Y 470.153,Z 479.213,A -85,B 0,C 180,E1 10793.957,E2 10793.957} C_VEL
LIN {X 0,Y 473.057,Z 483.544,A -85,B 0,C 180,E1 10791.614,E2 10791.614} C_VEL
LIN {X 0,Y 474.382,Z 485.18,A -85,B 0,C 180,E1 10790.721,E2 10790.721} C_VEL
LIN {X 0,Y 478.119,Z 490.324,A -85,B 0,C 180,E1 10788.479,E2 10788.479} C_VEL
LIN {X 0,Y 482.327,Z 496.277,A -85,B 0,C 180,E1 10786.33,E2 10786.33} C_VEL
LIN {X 0,Y 486.414,Z 502.089,A -85,B 0,C 180,E1 10784.5,E2 10784.5} C_VEL
LIN {X 0,Y 493.913,Z 512.896,A -85,B 0,C 180,E1 10781.59,E2 10781.59} C_VEL
LIN {X 0,Y 499.371,Z 521.673,A -85,B 0,C 180,E1 10779.702,E2 10779.702} C_VEL
LIN {X 0,Y 505.397,Z 532.434,A -85,B 0,C 180,E1 10777.778,E2 10777.778} C_VEL
LIN {X 0,Y 490.169,Z 750.178,A -85,B 0,C 180,E1 10774.385,E2 10774.385} C_VEL
LIN {X 0,Y 484.8,Z 826.074,A -85,B 0,C 180,E1 10773.181,E2 10773.181} C_VEL
LIN {X 0,Y 481.369,Z 854.509,A -85,B 0,C 180,E1 10772.629,E2 10772.629} C_VEL
LIN {X 0,Y 477.111,Z 879.536,A -85,B 0,C 180,E1 10771.99,E2 10771.99} C_VEL
LIN {X 0,Y 472.795,Z 900.791,A -85,B 0,C 180,E1 10771.31,E2 10771.31} C_VEL
LIN {X 0,Y 467.838,Z 921.815,A -85,B 0,C 180,E1 10770.504,E2 10770.504} C_VEL
LIN {X 0,Y 461.287,Z 946.323,A -85,B 0,C 180,E1 10769.377,E2 10769.377} C_VEL
LIN {X 0,Y 453.819,Z 970.472,A -85,B 0,C 180,E1 10768.023,E2 10768.023} C_VEL
LIN {X 0,Y 446.884,Z 990.763,A -85,B 0,C 180,E1 10766.688,E2 10766.688} C_VEL
LIN {X 0,Y 439.9,Z 1009.735,A -85,B 0,C 180,E1 10765.242,E2 10765.242} C_VEL
LIN {X 0,Y 432.423,Z 1028.728,A -85,B 0,C 180,E1 10763.579,E2 10763.579} C_VEL
LIN {X 0,Y 422.445,Z 1052.287,A -85,B 0,C 180,E1 10761.154,E2 10761.154} C_VEL
LIN {X 0,Y 414.564,Z 1069.88,A -85,B 0,C 180,E1 10759.019,E2 10759.019} C_VEL
LIN {X 0,Y 407.447,Z 1085.26,A -85,B 0,C 180,E1 10756.886,E2 10756.886} C_VEL
LIN {X 0,Y 400.052,Z 1100.892,A -85,B 0,C 180,E1 10754.413,E2 10754.413} C_VEL
LIN {X 0,Y 391.31,Z 1119.112,A -85,B 0,C 180,E1 10751.048,E2 10751.048} C_VEL
LIN {X 0,Y 384.667,Z 1132.962,A -85,B 0,C 180,E1 10748.028,E2 10748.028} C_VEL
LIN {X 0,Y 379.17,Z 1144.71,A -85,B 0,C 180,E1 10745.091,E2 10745.091} C_VEL
LIN {X 0,Y 374.206,Z 1155.701,A -85,B 0,C 180,E1 10741.942,E2 10741.942} C_VEL
LIN {X 0,Y 369.234,Z 1167.68,A -85,B 0,C 180,E1 10737.936,E2 10737.936} C_VEL
LIN {X 0,Y 365.568,Z 1177.346,A -85,B 0,C 180,E1 10733.999,E2 10733.999} C_VEL
LIN {X 0,Y 363.319,Z 1184.342,A -85,B 0,C 180,E1 10730.626,E2 10730.626} C_VEL
LIN {X 0,Y 361.708,Z 1190.285,A -85,B 0,C 180,E1 10727.205,E2 10727.205} C_VEL
LIN {X 0,Y 360.722,Z 1195.114,A -85,B 0,C 180,E1 10723.792,E2 10723.792} C_VEL
LIN {X 0,Y 360.159,Z 1199.187,A -85,B 0,C 180,E1 10720.073,E2 10720.073} C_VEL
LIN {X 0,Y 359.943,Z 1202.264,A -85,B 0,C 180,E1 10715.9,E2 10715.9} C_VEL
LIN {X 0,Y 359.913,Z 1203.608,A -85,B 0,C 180,E1 10712.23,E2 10712.23} C_VEL
LIN {X 0,Y 359.913,Z 1203.804,A -85,B 0,C 180,E1 10708.886,E2 10708.886} C_VEL
LIN {X 0,Y 359.919,Z 1202.994,A -85,B 0,C 180,E1 10705.539,E2 10705.539} C_VEL
LIN {X 0,Y 360,Z 1201.295,A -85,B 0,C 180,E1 10702.339,E2 10702.339} C_VEL
LIN {X 0,Y 360.263,Z 1198.519,A -85,B 0,C 180,E1 10698.96,E2 10698.96} C_VEL
LIN {X 0,Y 360.893,Z 1194.719,A -85,B 0,C 180,E1 10695.562,E2 10695.562} C_VEL
LIN {X 0,Y 361.928,Z 1190.131,A -85,B 0,C 180,E1 10692.309,E2 10692.309} C_VEL
LIN {X 0,Y 363.661,Z 1184.263,A -85,B 0,C 180,E1 10688.889,E2 10688.889} C_VEL
LIN {X 0,Y 366.248,Z 1176.934,A -85,B 0,C 180,E1 10685.311,E2 10685.311} C_VEL
LIN {X 0,Y 370.733,Z 1166.098,A -85,B 0,C 180,E1 10680.91,E2 10680.91} C_VEL
LIN {X 0,Y 375.895,Z 1154.834,A -85,B 0,C 180,E1 10677.137,E2 10677.137} C_VEL
LIN {X 0,Y 381.18,Z 1144.044,A -85,B 0,C 180,E1 10674.016,E2 10674.016} C_VEL
LIN {X 0,Y 387.72,Z 1131.303,A -85,B 0,C 180,E1 10670.816,E2 10670.816} C_VEL
LIN {X 0,Y 396.819,Z 1113.954,A -85,B 0,C 180,E1 10667.132,E2 10667.132} C_VEL
LIN {X 0,Y 404.632,Z 1098.967,A -85,B 0,C 180,E1 10664.428,E2 10664.428} C_VEL
LIN {X 0,Y 412.066,Z 1084.567,A -85,B 0,C 180,E1 10662.159,E2 10662.159} C_VEL
LIN {X 0,Y 419.575,Z 1069.685,A -85,B 0,C 180,E1 10660.097,E2 10660.097} C_VEL
LIN {X 0,Y 427.841,Z 1052.743,A -85,B 0,C 180,E1 10658.041,E2 10658.041} C_VEL
LIN {X 0,Y 438.328,Z 1030.107,A -85,B 0,C 180,E1 10655.702,E2 10655.702} C_VEL
LIN {X 0,Y 446.733,Z 1010.542,A -85,B 0,C 180,E1 10653.993,E2 10653.993} C_VEL
LIN {X 0,Y 454.34,Z 991.566,A -85,B 0,C 180,E1 10652.556,E2 10652.556} C_VEL
LIN {X 0,Y 461.573,Z 972.139,A -85,B 0,C 180,E1 10651.288,E2 10651.288} C_VEL
LIN {X 0,Y 469.028,Z 950.203,A -85,B 0,C 180,E1 10650.06,E2 10650.06} C_VEL
LIN {X 0,Y 476.969,Z 923.436,A -85,B 0,C 180,E1 10648.827,E2 10648.827} C_VEL
LIN {X 0,Y 482.484,Z 901.978,A -85,B 0,C 180,E1 10648.017,E2 10648.017} C_VEL
LIN {X 0,Y 487.194,Z 880.735,A -85,B 0,C 180,E1 10647.351,E2 10647.351} C_VEL
LIN {X 0,Y 491.266,Z 858.946,A -85,B 0,C 180,E1 10646.799,E2 10646.799} C_VEL
LIN {X 0,Y 495.268,Z 831.434,A -85,B 0,C 180,E1 10646.248,E2 10646.248} C_VEL
LIN {X 0,Y 499.077,Z 786.094,A -85,B 0,C 180,E1 10645.519,E2 10645.519} C_VEL
LIN {X 0,Y 516.367,Z 565.569,A -85,B 0,C 180,E1 10642.097,E2 10642.097} C_VEL
LIN {X 0,Y 518.487,Z 538.971,A -85,B 0,C 180,E1 10641.673,E2 10641.673} C_VEL
LIN {X 0,Y 512.971,Z 529.27,A -85,B 0,C 180,E1 10639.352,E2 10639.352} C_VEL
LIN {X 0,Y 507.765,Z 521.262,A -85,B 0,C 180,E1 10636.826,E2 10636.826} C_VEL
LIN {X 0,Y 504.086,Z 515.927,A -85,B 0,C 180,E1 10634.708,E2 10634.708} C_VEL
LIN {X 0,Y 501.169,Z 511.597,A -85,B 0,C 180,E1 10632.678,E2 10632.678} C_VEL
LIN {X 0,Y 498.364,Z 507.352,A -85,B 0,C 180,E1 10630.169,E2 10630.169} C_VEL
LIN {X 0,Y 497.733,Z 506.474,A -85,B 0,C 180,E1 10629.481,E2 10629.481} C_VEL
LIN {X 0,Y 495.13,Z 502.388,A -85,B 0,C 180,E1 10624.633,E2 10624.633} C_VEL
LIN {X 0,Y 495.053,Z 501.086,A -85,B 0,C 180,E1 10623.01,E2 10623.01} C_VEL
LIN {X 0,Y 495.068,Z 501.681,A -85,B 0,C 180,E1 10621.852,E2 10621.852} C_VEL
LIN {X 0,Y 497.526,Z 506.282,A -85,B 0,C 180,E1 10616.543,E2 10616.543} C_VEL
LIN {X 0,Y 498.259,Z 507.147,A -85,B 0,C 180,E1 10615.742,E2 10615.742} C_VEL
LIN {X 0,Y 501.916,Z 512.682,A -85,B 0,C 180,E1 10612.56,E2 10612.56} C_VEL
LIN {X 0,Y 505.544,Z 517.978,A -85,B 0,C 180,E1 10610.207,E2 10610.207} C_VEL
LIN {X 0,Y 508.996,Z 523.202,A -85,B 0,C 180,E1 10608.326,E2 10608.326} C_VEL
LIN {X 0,Y 514.103,Z 530.828,A -85,B 0,C 180,E1 10605.958,E2 10605.958} C_VEL
LIN {X 0,Y 518.489,Z 537.955,A -85,B 0,C 180,E1 10604.164,E2 10604.164} C_VEL
LIN {X 0,Y 502.141,Z 744.284,A -85,B 0,C 180,E1 10600.964,E2 10600.964} C_VEL
LIN {X 0,Y 496.011,Z 821.28,A -85,B 0,C 180,E1 10599.749,E2 10599.749} C_VEL
LIN {X 0,Y 492.315,Z 849.67,A -85,B 0,C 180,E1 10599.207,E2 10599.207} C_VEL
LIN {X 0,Y 487.803,Z 874.506,A -85,B 0,C 180,E1 10598.581,E2 10598.581} C_VEL
LIN {X 0,Y 483.336,Z 895.051,A -85,B 0,C 180,E1 10597.936,E2 10597.936} C_VEL
LIN {X 0,Y 478.16,Z 915.576,A -85,B 0,C 180,E1 10597.167,E2 10597.167} C_VEL
LIN {X 0,Y 472.044,Z 936.952,A -85,B 0,C 180,E1 10596.212,E2 10596.212} C_VEL
LIN {X 0,Y 463.525,Z 963.073,A -85,B 0,C 180,E1 10594.81,E2 10594.81} C_VEL
LIN {X 0,Y 455.583,Z 984.555,A -85,B 0,C 180,E1 10593.423,E2 10593.423} C_VEL
LIN {X 0,Y 447.945,Z 1003.666,A -85,B 0,C 180,E1 10591.982,E2 10591.982} C_VEL
LIN {X 0,Y 440.282,Z 1021.538,A -85,B 0,C 180,E1 10590.433,E2 10590.433} C_VEL
LIN {X 0,Y 430.655,Z 1042.702,A -85,B 0,C 180,E1 10588.311,E2 10588.311} C_VEL
LIN {X 0,Y 421.044,Z 1062.253,A -85,B 0,C 180,E1 10585.973,E2 10585.973} C_VEL
LIN {X 0,Y 412.866,Z 1078.31,A -85,B 0,C 180,E1 10583.75,E2 10583.75} C_VEL
LIN {X 0,Y 405.283,Z 1092.824,A -85,B 0,C 180,E1 10581.45,E2 10581.45} C_VEL
LIN {X 0,Y 397.463,Z 1107.587,A -85,B 0,C 180,E1 10578.768,E2 10578.768} C_VEL
LIN {X 0,Y 388.289,Z 1124.788,A -85,B 0,C 180,E1 10575.083,E2 10575.083} C_VEL
LIN {X 0,Y 381.739,Z 1137.307,A -85,B 0,C 180,E1 10571.905,E2 10571.905} C_VEL
LIN {X 0,Y 376.411,Z 1147.861,A -85,B 0,C 180,E1 10568.821,E2 10568.821} C_VEL
LIN {X 0,Y 371.522,Z 1158.128,A -85,B 0,C 180,E1 10565.353,E2 10565.353} C_VEL
LIN {X 0,Y 366.688,Z 1169.335,A -85,B 0,C 180,E1 10560.801,E2 10560.801} C_VEL
LIN {X 0,Y 363.923,Z 1176.745,A -85,B 0,C 180,E1 10557.134,E2 10557.134} C_VEL
LIN {X 0,Y 362.159,Z 1182.425,A -85,B 0,C 180,E1 10553.771,E2 10553.771} C_VEL
LIN {X 0,Y 361.011,Z 1187.064,A -85,B 0,C 180,E1 10550.424,E2 10550.424} C_VEL
LIN {X 0,Y 360.36,Z 1190.7,A -85,B 0,C 180,E1 10547.104,E2 10547.104} C_VEL
LIN {X 0,Y 360.046,Z 1193.367,A -85,B 0,C 180,E1 10543.817,E2 10543.817} C_VEL
LIN {X 0,Y 359.935,Z 1195.092,A -85,B 0,C 180,E1 10540.564,E2 10540.564} C_VEL
LIN {X 0,Y 359.922,Z 1195.895,A -85,B 0,C 180,E1 10537.341,E2 10537.341} C_VEL
LIN {X 0,Y 359.916,Z 1195.792,A -85,B 0,C 180,E1 10534.141,E2 10534.141} C_VEL
LIN {X 0,Y 359.94,Z 1194.795,A -85,B 0,C 180,E1 10530.954,E2 10530.954} C_VEL
LIN {X 0,Y 360.055,Z 1192.907,A -85,B 0,C 180,E1 10527.771,E2 10527.771} C_VEL
LIN {X 0,Y 360.381,Z 1189.969,A -85,B 0,C 180,E1 10524.427,E2 10524.427} C_VEL
LIN {X 0,Y 361.221,Z 1185.427,A -85,B 0,C 180,E1 10520.6,E2 10520.6} C_VEL
LIN {X 0,Y 363.065,Z 1178.332,A -85,B 0,C 180,E1 10516.137,E2 10516.137} C_VEL
LIN {X 0,Y 365.304,Z 1171.429,A -85,B 0,C 180,E1 10512.641,E2 10512.641} C_VEL
LIN {X 0,Y 368.188,Z 1163.7,A -85,B 0,C 180,E1 10509.326,E2 10509.326} C_VEL
LIN {X 0,Y 371.886,Z 1154.786,A -85,B 0,C 180,E1 10506.046,E2 10506.046} C_VEL
LIN {X 0,Y 373.858,Z 1150.337,A -85,B 0,C 180,E1 10504.561,E2 10504.561} C_VEL
LIN {X 0,Y 374.375,Z 1147.136,A -85,B 0,C 180,E1 10503.485,E2 10503.485} C_VEL
LIN {X 0,Y 372.888,Z 1138.728,A -85,B 0,C 180,E1 10500.5,E2 10500.5} C_VEL
LIN {X 0,Y 373.749,Z 1135.663,A -85,B 0,C 180,E1 10499.598,E2 10499.598} C_VEL
LIN {X 0,Y 381.754,Z 1119.775,A -85,B 0,C 180,E1 10495.728,E2 10495.728} C_VEL
LIN {X 0,Y 388.878,Z 1105.674,A -85,B 0,C 180,E1 10492.826,E2 10492.826} C_VEL
LIN {X 0,Y 395.99,Z 1091.554,A -85,B 0,C 180,E1 10490.295,E2 10490.295} C_VEL
LIN {X 0,Y 403.733,Z 1075.888,A -85,B 0,C 180,E1 10487.843,E2 10487.843} C_VEL
LIN {X 0,Y 413.553,Z 1055.317,A -85,B 0,C 180,E1 10485.09,E2 10485.09} C_VEL
LIN {X 0,Y 421.829,Z 1036.951,A -85,B 0,C 180,E1 10483.008,E2 10483.008} C_VEL
LIN {X 0,Y 429.236,Z 1019.661,A -85,B 0,C 180,E1 10481.301,E2 10481.301} C_VEL
LIN {X 0,Y 436.394,Z 1001.876,A -85,B 0,C 180,E1 10479.762,E2 10479.762} C_VEL
LIN {X 0,Y 444.129,Z 981.256,A -85,B 0,C 180,E1 10478.213,E2 10478.213} C_VEL
LIN {X 0,Y 452.767,Z 955.687,A -85,B 0,C 180,E1 10476.603,E2 10476.603} C_VEL
LIN {X 0,Y 459.202,Z 934.248,A -85,B 0,C 180,E1 10475.476,E2 10475.476} C_VEL
LIN {X 0,Y 464.627,Z 914.014,A -85,B 0,C 180,E1 10474.569,E2 10474.569} C_VEL
LIN {X 0,Y 469.534,Z 893.223,A -85,B 0,C 180,E1 10473.781,E2 10473.781} C_VEL
LIN {X 0,Y 474.767,Z 867.222,A -85,B 0,C 180,E1 10472.972,E2 10472.972} C_VEL
LIN {X 0,Y 478.895,Z 840.24,A -85,B 0,C 180,E1 10472.341,E2 10472.341} C_VEL
LIN {X 0,Y 481.428,Z 817.637,A -85,B 0,C 180,E1 10471.925,E2 10471.925} C_VEL
LIN {X 0,Y 496.649,Z 605.092,A -85,B 0,C 180,E1 10468.598,E2 10468.598} C_VEL
LIN {X 0,Y 501.633,Z 535.503,A -85,B 0,C 180,E1 10467.487,E2 10467.487} C_VEL
LIN {X 0,Y 494.336,Z 523.949,A -85,B 0,C 180,E1 10465.072,E2 10465.072} C_VEL
LIN {X 0,Y 487.128,Z 513.04,A -85,B 0,C 180,E1 10462.349,E2 10462.349} C_VEL
LIN {X 0,Y 481.927,Z 505.431,A -85,B 0,C 180,E1 10460.083,E2 10460.083} C_VEL
LIN {X 0,Y 478.613,Z 500.749,A -85,B 0,C 180,E1 10458.452,E2 10458.452} C_VEL
LIN {X 0,Y 475.535,Z 496.361,A -85,B 0,C 180,E1 10456.742,E2 10456.742} C_VEL
LIN {X 0,Y 472.214,Z 491.651,A -85,B 0,C 180,E1 10454.595,E2 10454.595} C_VEL
LIN {X 0,Y 469.108,Z 487.323,A -85,B 0,C 180,E1 10452.119,E2 10452.119} C_VEL
LIN {X 0,Y 468.406,Z 486.305,A -85,B 0,C 180,E1 10451.451,E2 10451.451} C_VEL
LIN {X 0,Y 465.83,Z 483.188,A -85,B 0,C 180,E1 10448.393,E2 10448.393} C_VEL
LIN {X 0,Y 465.023,Z 480.946,A -85,B 0,C 180,E1 10446.668,E2 10446.668} C_VEL
LIN {X 0,Y 464.588,Z 480.781,A -85,B 0,C 180,E1 10440.493,E2 10440.493} C_VEL
LIN {X 0,Y 465.156,Z 481.143,A -85,B 0,C 180,E1 10439.138,E2 10439.138} C_VEL
LIN {X 0,Y 466.812,Z 484.858,A -85,B 0,C 180,E1 10436.316,E2 10436.316} C_VEL
LIN {X 0,Y 469.026,Z 487.152,A -85,B 0,C 180,E1 10434.065,E2 10434.065} C_VEL
LIN {X 0,Y 472.077,Z 491.593,A -85,B 0,C 180,E1 10431.596,E2 10431.596} C_VEL
LIN {X 0,Y 473.466,Z 493.592,A -85,B 0,C 180,E1 10430.641,E2 10430.641} C_VEL
LIN {X 0,Y 476.596,Z 497.852,A -85,B 0,C 180,E1 10428.749,E2 10428.749} C_VEL
LIN {X 0,Y 480.96,Z 504.165,A -85,B 0,C 180,E1 10426.474,E2 10426.474} C_VEL
LIN {X 0,Y 486.091,Z 511.481,A -85,B 0,C 180,E1 10424.184,E2 10424.184} C_VEL
LIN {X 0,Y 492.958,Z 521.848,A -85,B 0,C 180,E1 10421.523,E2 10421.523} C_VEL
LIN {X 0,Y 497.663,Z 529.722,A -85,B 0,C 180,E1 10419.875,E2 10419.875} C_VEL
LIN {X 0,Y 501.725,Z 537.186,A -85,B 0,C 180,E1 10418.536,E2 10418.536} C_VEL
LIN {X 0,Y 486.017,Z 756.079,A -85,B 0,C 180,E1 10415.126,E2 10415.126} C_VEL
LIN {X 0,Y 480.883,Z 826.398,A -85,B 0,C 180,E1 10414.008,E2 10414.008} C_VEL
LIN {X 0,Y 477.224,Z 855.61,A -85,B 0,C 180,E1 10413.439,E2 10413.439} C_VEL
LIN {X 0,Y 473.019,Z 879.76,A -85,B 0,C 180,E1 10412.822,E2 10412.822} C_VEL
LIN {X 0,Y 468.569,Z 901.167,A -85,B 0,C 180,E1 10412.139,E2 10412.139} C_VEL
LIN {X 0,Y 463.504,Z 922.138,A -85,B 0,C 180,E1 10411.336,E2 10411.336} C_VEL
LIN {X 0,Y 456.75,Z 946.806,A -85,B 0,C 180,E1 10410.202,E2 10410.202} C_VEL
LIN {X 0,Y 448.85,Z 971.594,A -85,B 0,C 180,E1 10408.806,E2 10408.806} C_VEL
LIN {X 0,Y 442.063,Z 990.943,A -85,B 0,C 180,E1 10407.53,E2 10407.53} C_VEL
LIN {X 0,Y 434.934,Z 1009.815,A -85,B 0,C 180,E1 10406.09,E2 10406.09} C_VEL
LIN {X 0,Y 426.948,Z 1029.54,A -85,B 0,C 180,E1 10404.356,E2 10404.356} C_VEL
LIN {X 0,Y 416.732,Z 1052.891,A -85,B 0,C 180,E1 10401.929,E2 10401.929} C_VEL
LIN {X 0,Y 408.847,Z 1069.966,A -85,B 0,C 180,E1 10399.841,E2 10399.841} C_VEL
LIN {X 0,Y 401.516,Z 1085.305,A -85,B 0,C 180,E1 10397.698,E2 10397.698} C_VEL
LIN {X 0,Y 394.062,Z 1100.526,A -85,B 0,C 180,E1 10395.273,E2 10395.273} C_VEL
LIN {X 0,Y 385.345,Z 1118.08,A -85,B 0,C 180,E1 10392.025,E2 10392.025} C_VEL
LIN {X 0,Y 378.031,Z 1132.673,A -85,B 0,C 180,E1 10388.819,E2 10388.819} C_VEL
LIN {X 0,Y 372.158,Z 1144.705,A -85,B 0,C 180,E1 10385.767,E2 10385.767} C_VEL
LIN {X 0,Y 366.85,Z 1155.982,A -85,B 0,C 180,E1 10382.476,E2 10382.476} C_VEL
LIN {X 0,Y 361.477,Z 1168.297,A -85,B 0,C 180,E1 10378.23,E2 10378.23} C_VEL
LIN {X 0,Y 357.871,Z 1177.41,A -85,B 0,C 180,E1 10374.426,E2 10374.426} C_VEL
LIN {X 0,Y 355.471,Z 1184.478,A -85,B 0,C 180,E1 10370.931,E2 10370.931} C_VEL
LIN {X 0,Y 353.786,Z 1190.388,A -85,B 0,C 180,E1 10367.433,E2 10367.433} C_VEL
LIN {X 0,Y 352.754,Z 1195.184,A -85,B 0,C 180,E1 10363.942,E2 10363.942} C_VEL
LIN {X 0,Y 352.135,Z 1199.547,A -85,B 0,C 180,E1 10359.81,E2 10359.81} C_VEL
LIN {X 0,Y 351.939,Z 1202.298,A -85,B 0,C 180,E1 10355.707,E2 10355.707} C_VEL
LIN {X 0,Y 351.913,Z 1203.538,A -85,B 0,C 180,E1 10352.117,E2 10352.117} C_VEL
LIN {X 0,Y 351.914,Z 1203.722,A -85,B 0,C 180,E1 10348.861,E2 10348.861} C_VEL
LIN {X 0,Y 351.92,Z 1202.922,A -85,B 0,C 180,E1 10345.438,E2 10345.438} C_VEL
LIN {X 0,Y 352.006,Z 1201.234,A -85,B 0,C 180,E1 10342.164,E2 10342.164} C_VEL
LIN {X 0,Y 352.291,Z 1198.468,A -85,B 0,C 180,E1 10338.707,E2 10338.707} C_VEL
LIN {X 0,Y 352.976,Z 1194.682,A -85,B 0,C 180,E1 10335.23,E2 10335.23} C_VEL
LIN {X 0,Y 354.172,Z 1189.853,A -85,B 0,C 180,E1 10331.738,E2 10331.738} C_VEL
LIN {X 0,Y 356.05,Z 1183.95,A -85,B 0,C 180,E1 10328.243,E2 10328.243} C_VEL
LIN {X 0,Y 358.999,Z 1176.238,A -85,B 0,C 180,E1 10324.425,E2 10324.425} C_VEL
LIN {X 0,Y 363.997,Z 1164.895,A -85,B 0,C 180,E1 10319.823,E2 10319.823} C_VEL
LIN {X 0,Y 368.878,Z 1154.898,A -85,B 0,C 180,E1 10316.431,E2 10316.431} C_VEL
LIN {X 0,Y 374.477,Z 1144.015,A -85,B 0,C 180,E1 10313.229,E2 10313.229} C_VEL
LIN {X 0,Y 380.912,Z 1132.042,A -85,B 0,C 180,E1 10310.173,E2 10310.173} C_VEL
LIN {X 0,Y 389.932,Z 1115.64,A -85,B 0,C 180,E1 10306.591,E2 10306.591} C_VEL
LIN {X 0,Y 398.837,Z 1099.153,A -85,B 0,C 180,E1 10303.572,E2 10303.572} C_VEL
LIN {X 0,Y 406.876,Z 1084.135,A -85,B 0,C 180,E1 10301.194,E2 10301.194} C_VEL
LIN {X 0,Y 415.071,Z 1068.433,A -85,B 0,C 180,E1 10299.025,E2 10299.025} C_VEL
LIN {X 0,Y 425.323,Z 1048.074,A -85,B 0,C 180,E1 10296.601,E2 10296.601} C_VEL
LIN {X 0,Y 435.352,Z 1026.526,A -85,B 0,C 180,E1 10294.461,E2 10294.461} C_VEL
LIN {X 0,Y 443.213,Z 1008.649,A -85,B 0,C 180,E1 10292.936,E2 10292.936} C_VEL
LIN {X 0,Y 450.701,Z 990.371,A -85,B 0,C 180,E1 10291.572,E2 10291.572} C_VEL
LIN {X 0,Y 458.508,Z 969.779,A -85,B 0,C 180,E1 10290.249,E2 10290.249} C_VEL
LIN {X 0,Y 467.416,Z 943.493,A -85,B 0,C 180,E1 10288.84,E2 10288.84} C_VEL
LIN {X 0,Y 473.917,Z 921.514,A -85,B 0,C 180,E1 10287.871,E2 10287.871} C_VEL
LIN {X 0,Y 479.327,Z 900.741,A -85,B 0,C 180,E1 10287.103,E2 10287.103} C_VEL
LIN {X 0,Y 484.205,Z 879.017,A -85,B 0,C 180,E1 10286.438,E2 10286.438} C_VEL
LIN {X 0,Y 488.8,Z 854.427,A -85,B 0,C 180,E1 10285.837,E2 10285.837} C_VEL
LIN {X 0,Y 492.628,Z 825.865,A -85,B 0,C 180,E1 10285.3,E2 10285.3} C_VEL
LIN {X 0,Y 498.803,Z 750.14,A -85,B 0,C 180,E1 10284.107,E2 10284.107} C_VEL
LIN {X 0,Y 515.491,Z 544.249,A -85,B 0,C 180,E1 10280.919,E2 10280.919} C_VEL
LIN {X 0,Y 511.014,Z 536.291,A -85,B 0,C 180,E1 10278.954,E2 10278.954} C_VEL
LIN {X 0,Y 506.057,Z 528.567,A -85,B 0,C 180,E1 10276.471,E2 10276.471} C_VEL
LIN {X 0,Y 502.666,Z 523.515,A -85,B 0,C 180,E1 10274.456,E2 10274.456} C_VEL
LIN {X 0,Y 499.898,Z 519.333,A -85,B 0,C 180,E1 10272.475,E2 10272.475} C_VEL
LIN {X 0,Y 497.177,Z 515.052,A -85,B 0,C 180,E1 10269.96,E2 10269.96} C_VEL
LIN {X 0,Y 496.064,Z 513.865,A -85,B 0,C 180,E1 10268.695,E2 10268.695} C_VEL
LIN {X 0,Y 494.077,Z 509.027,A -85,B 0,C 180,E1 10263.016,E2 10263.016} C_VEL
LIN {X 0,Y 494.106,Z 509.84,A -85,B 0,C 180,E1 10261.623,E2 10261.623} C_VEL
LIN {X 0,Y 496.446,Z 514.164,A -85,B 0,C 180,E1 10256.651,E2 10256.651} C_VEL
LIN {X 0,Y 497.162,Z 515.059,A -85,B 0,C 180,E1 10255.848,E2 10255.848} C_VEL
LIN {X 0,Y 500.617,Z 520.357,A -85,B 0,C 180,E1 10252.771,E2 10252.771} C_VEL
LIN {X 0,Y 504.167,Z 525.661,A -85,B 0,C 180,E1 10250.41,E2 10250.41} C_VEL
LIN {X 0,Y 507.663,Z 531.071,A -85,B 0,C 180,E1 10248.468,E2 10248.468} C_VEL
LIN {X 0,Y 512.462,Z 538.38,A -85,B 0,C 180,E1 10246.2,E2 10246.2} C_VEL
LIN {X 0,Y 515.449,Z 543.505,A -85,B 0,C 180,E1 10244.923,E2 10244.923} C_VEL
LIN {X 0,Y 498.669,Z 750.253,A -85,B 0,C 180,E1 10241.724,E2 10241.724} C_VEL
LIN {X 0,Y 492.817,Z 821.651,A -85,B 0,C 180,E1 10240.599,E2 10240.599} C_VEL
LIN {X 0,Y 488.967,Z 850.374,A -85,B 0,C 180,E1 10240.051,E2 10240.051} C_VEL
LIN {X 0,Y 484.451,Z 874.707,A -85,B 0,C 180,E1 10239.442,E2 10239.442} C_VEL
LIN {X 0,Y 479.902,Z 895.191,A -85,B 0,C 180,E1 10238.805,E2 10238.805} C_VEL
LIN {X 0,Y 474.618,Z 915.696,A -85,B 0,C 180,E1 10238.042,E2 10238.042} C_VEL
LIN {X 0,Y 468.367,Z 937.061,A -85,B 0,C 180,E1 10237.096,E2 10237.096} C_VEL
LIN {X 0,Y 459.653,Z 963.175,A -85,B 0,C 180,E1 10235.704,E2 10235.704} C_VEL
LIN {X 0,Y 451.525,Z 984.644,A -85,B 0,C 180,E1 10234.325,E2 10234.325} C_VEL
LIN {X 0,Y 443.95,Z 1003.147,A -85,B 0,C 180,E1 10232.938,E2 10232.938} C_VEL
LIN {X 0,Y 436.433,Z 1020.243,A -85,B 0,C 180,E1 10231.473,E2 10231.473} C_VEL
LIN {X 0,Y 427.938,Z 1038.41,A -85,B 0,C 180,E1 10229.689,E2 10229.689} C_VEL
LIN {X 0,Y 417.306,Z 1059.848,A -85,B 0,C 180,E1 10227.213,E2 10227.213} C_VEL
LIN {X 0,Y 408.276,Z 1077.018,A -85,B 0,C 180,E1 10224.863,E2 10224.863} C_VEL
LIN {X 0,Y 400.391,Z 1091.582,A -85,B 0,C 180,E1 10222.571,E2 10222.571} C_VEL
LIN {X 0,Y 392.832,Z 1105.305,A -85,B 0,C 180,E1 10220.102,E2 10220.102} C_VEL
LIN {X 0,Y 384.823,Z 1119.793,A -85,B 0,C 180,E1 10217.097,E2 10217.097} C_VEL
LIN {X 0,Y 376.201,Z 1135.401,A -85,B 0,C 180,E1 10213.259,E2 10213.259} C_VEL
LIN {X 0,Y 370.205,Z 1146.604,A -85,B 0,C 180,E1 10210.001,E2 10210.001} C_VEL
LIN {X 0,Y 365.377,Z 1156.082,A -85,B 0,C 180,E1 10206.819,E2 10206.819} C_VEL
LIN {X 0,Y 361.235,Z 1164.822,A -85,B 0,C 180,E1 10203.422,E2 10203.422} C_VEL
LIN {X 0,Y 357.326,Z 1174.173,A -85,B 0,C 180,E1 10199.136,E2 10199.136} C_VEL
LIN {X 0,Y 354.575,Z 1181.85,A -85,B 0,C 180,E1 10194.667,E2 10194.667} C_VEL
LIN {X 0,Y 353.243,Z 1186.615,A -85,B 0,C 180,E1 10191.242,E2 10191.242} C_VEL
LIN {X 0,Y 352.469,Z 1190.374,A -85,B 0,C 180,E1 10187.84,E2 10187.84} C_VEL
LIN {X 0,Y 352.104,Z 1193.047,A -85,B 0,C 180,E1 10184.639,E2 10184.639} C_VEL
LIN {X 0,Y 351.95,Z 1194.936,A -85,B 0,C 180,E1 10181.304,E2 10181.304} C_VEL
LIN {X 0,Y 351.923,Z 1195.88,A -85,B 0,C 180,E1 10178.166,E2 10178.166} C_VEL
LIN {X 0,Y 351.907,Z 1195.984,A -85,B 0,C 180,E1 10174.889,E2 10174.889} C_VEL
LIN {X 0,Y 351.931,Z 1195.192,A -85,B 0,C 180,E1 10171.627,E2 10171.627} C_VEL
LIN {X 0,Y 352.026,Z 1193.509,A -85,B 0,C 180,E1 10168.372,E2 10168.372} C_VEL
LIN {X 0,Y 352.31,Z 1190.813,A -85,B 0,C 180,E1 10164.989,E2 10164.989} C_VEL
LIN {X 0,Y 352.938,Z 1187.253,A -85,B 0,C 180,E1 10161.692,E2 10161.692} C_VEL
LIN {X 0,Y 354.044,Z 1182.556,A -85,B 0,C 180,E1 10158.267,E2 10158.267} C_VEL
LIN {X 0,Y 355.787,Z 1176.815,A -85,B 0,C 180,E1 10154.849,E2 10154.849} C_VEL
LIN {X 0,Y 358.357,Z 1169.65,A -85,B 0,C 180,E1 10151.284,E2 10151.284} C_VEL
LIN {X 0,Y 362.715,Z 1159.157,A -85,B 0,C 180,E1 10146.955,E2 10146.955} C_VEL
LIN {X 0,Y 367.523,Z 1148.506,A -85,B 0,C 180,E1 10143.327,E2 10143.327} C_VEL
LIN {X 0,Y 372.606,Z 1137.989,A -85,B 0,C 180,E1 10140.235,E2 10140.235} C_VEL
LIN {X 0,Y 373.749,Z 1135.663,A -85,B 0,C 180,E1 10139.598,E2 10139.598} C_VEL
LIN {X 0,Y 374.722,Z 1132.11,A -85,B 0,C 180,E1 10138.552,E2 10138.552} C_VEL
LIN {X 0,Y 374.437,Z 1122.648,A -85,B 0,C 180,E1 10135.643,E2 10135.643} C_VEL
LIN {X 0,Y 375.605,Z 1119.162,A -85,B 0,C 180,E1 10134.794,E2 10134.794} C_VEL
LIN {X 0,Y 382.818,Z 1105.417,A -85,B 0,C 180,E1 10131.945,E2 10131.945} C_VEL
LIN {X 0,Y 389.779,Z 1092.079,A -85,B 0,C 180,E1 10129.533,E2 10129.533} C_VEL
LIN {X 0,Y 396.843,Z 1078.258,A -85,B 0,C 180,E1 10127.33,E2 10127.33} C_VEL
LIN {X 0,Y 404.652,Z 1062.546,A -85,B 0,C 180,E1 10125.133,E2 10125.133} C_VEL
LIN {X 0,Y 414.552,Z 1041.8,A -85,B 0,C 180,E1 10122.638,E2 10122.638} C_VEL
LIN {X 0,Y 423.425,Z 1021.735,A -85,B 0,C 180,E1 10120.609,E2 10120.609} C_VEL
LIN {X 0,Y 431.034,Z 1003.408,A -85,B 0,C 180,E1 10119.003,E2 10119.003} C_VEL
LIN {X 0,Y 438.34,Z 984.511,A -85,B 0,C 180,E1 10117.564,E2 10117.564} C_VEL
LIN {X 0,Y 446.541,Z 961.523,A -85,B 0,C 180,E1 10116.066,E2 10116.066} C_VEL
LIN {X 0,Y 454.349,Z 936.503,A -85,B 0,C 180,E1 10114.716,E2 10114.716} C_VEL
LIN {X 0,Y 460.171,Z 915.421,A -85,B 0,C 180,E1 10113.763,E2 10113.763} C_VEL
LIN {X 0,Y 465.163,Z 894.879,A -85,B 0,C 180,E1 10112.981,E2 10112.981} C_VEL
LIN {X 0,Y 469.739,Z 872.902,A -85,B 0,C 180,E1 10112.282,E2 10112.282} C_VEL
LIN {X 0,Y 474.47,Z 844.984,A -85,B 0,C 180,E1 10111.588,E2 10111.588} C_VEL
LIN {X 0,Y 477.497,Z 819.477,A -85,B 0,C 180,E1 10111.109,E2 10111.109} C_VEL
LIN {X 0,Y 490.789,Z 638.852,A -85,B 0,C 180,E1 10108.279,E2 10108.279} C_VEL
LIN {X 0,Y 498.063,Z 540.419,A -85,B 0,C 180,E1 10106.724,E2 10106.724} C_VEL
LIN {X 0,Y 490.945,Z 529.108,A -85,B 0,C 180,E1 10104.261,E2 10104.261} C_VEL
LIN {X 0,Y 484.046,Z 518.363,A -85,B 0,C 180,E1 10101.51,E2 10101.51} C_VEL
LIN {X 0,Y 477.879,Z 509.293,A -85,B 0,C 180,E1 10098.608,E2 10098.608} C_VEL
LIN {X 0,Y 473.962,Z 503.831,A -85,B 0,C 180,E1 10096.421,E2 10096.421} C_VEL
LIN {X 0,Y 470.901,Z 499.375,A -85,B 0,C 180,E1 10094.385,E2 10094.385} C_VEL
LIN {X 0,Y 467.813,Z 494.892,A -85,B 0,C 180,E1 10091.841,E2 10091.841} C_VEL
LIN {X 0,Y 466.683,Z 493.708,A -85,B 0,C 180,E1 10090.743,E2 10090.743} C_VEL
LIN {X 0,Y 464.338,Z 489.931,A -85,B 0,C 180,E1 10087.424,E2 10087.424} C_VEL
LIN {X 0,Y 463.994,Z 488.867,A -85,B 0,C 180,E1 10086.558,E2 10086.558} C_VEL
LIN {X 0,Y 463.653,Z 488.746,A -85,B 0,C 180,E1 10080.371,E2 10080.371} C_VEL
LIN {X 0,Y 464.161,Z 489.228,A -85,B 0,C 180,E1 10079.136,E2 10079.136} C_VEL
LIN {X 0,Y 465.831,Z 492.849,A -85,B 0,C 180,E1 10076.308,E2 10076.308} C_VEL
LIN {X 0,Y 467.841,Z 494.957,A -85,B 0,C 180,E1 10074.235,E2 10074.235} C_VEL
LIN {X 0,Y 470.75,Z 499.3,A -85,B 0,C 180,E1 10071.818,E2 10071.818} C_VEL
LIN {X 0,Y 472.376,Z 501.691,A -85,B 0,C 180,E1 10070.681,E2 10070.681} C_VEL
LIN {X 0,Y 475.183,Z 505.553,A -85,B 0,C 180,E1 10068.961,E2 10068.961} C_VEL
LIN {X 0,Y 479.478,Z 511.87,A -85,B 0,C 180,E1 10066.677,E2 10066.677} C_VEL
LIN {X 0,Y 484.337,Z 518.941,A -85,B 0,C 180,E1 10064.463,E2 10064.463} C_VEL
LIN {X 0,Y 491.02,Z 529.206,A -85,B 0,C 180,E1 10061.816,E2 10061.816} C_VEL
LIN {X 0,Y 495.488,Z 536.87,A -85,B 0,C 180,E1 10060.213,E2 10060.213} C_VEL
LIN {X 0,Y 498.147,Z 541.868,A -85,B 0,C 180,E1 10059.306,E2 10059.306} C_VEL
LIN {X 0,Y 481.897,Z 762.68,A -85,B 0,C 180,E1 10055.869,E2 10055.869} C_VEL
LIN {X 0,Y 477.069,Z 826.691,A -85,B 0,C 180,E1 10054.85,E2 10054.85} C_VEL
LIN {X 0,Y 473.176,Z 856.692,A -85,B 0,C 180,E1 10054.262,E2 10054.262} C_VEL
LIN {X 0,Y 469.034,Z 879.929,A -85,B 0,C 180,E1 10053.669,E2 10053.669} C_VEL
LIN {X 0,Y 464.574,Z 900.939,A -85,B 0,C 180,E1 10053.003,E2 10053.003} C_VEL
LIN {X 0,Y 459.44,Z 921.798,A -85,B 0,C 180,E1 10052.211,E2 10052.211} C_VEL
LIN {X 0,Y 452.428,Z 946.864,A -85,B 0,C 180,E1 10051.066,E2 10051.066} C_VEL
LIN {X 0,Y 444.604,Z 970.87,A -85,B 0,C 180,E1 10049.722,E2 10049.722} C_VEL
LIN {X 0,Y 437.339,Z 991.109,A -85,B 0,C 180,E1 10048.391,E2 10048.391} C_VEL
